(* CODESYS project CowbellCheckers_Rev8.project

Project tree, tasks and I/O mapping:
  CODESYS_SoftMotion_Win_V3 : PAC320-CXX2X-XX, Parker Hannifin, order no. PAC320-CXX2X-XX, version 3.5.9.10
    application Application
      libraries: VisuDialogs, * (System); CmpErrors, 3.3.1.40 (System); ISysTypes2, 3.5.0.0 (System); SysFile, 3.5.9.0 (System); SysTimeCore, 3.5.5.0 (System); SysTimeRtc, 3.5.5.0 (System); Util, 3.5.9.0 (System)
      task VISU_TASK (cyclic, interval 100 ms, priority 31) calls VisuElems.Visu_Prg
      task EtherCAT_Master_Sim (externalevent, external event EVENT_ECM_DC, priority 0) calls EtherCAT_Master.EtherCAT_Task [EtherCAT_Master.EtherCAT_Task], Gameplay, KingTextControl, TurnEnforcer, TestPower, MakeMove, AxisPositionFeedback, JogLogic, SetupStart, CheckForWinner, Teardown
      task FileHandler (cyclic, interval t#20ms, priority 25) calls LogData
      global variables GlobalVars
      SymbolConfiguration
      JogFunctionality/
        program JogLogic [ST]
      Visualizations/
        visualisation AreYouSure
        visualisation ErrorVis
        visualisation JogVis
        visualisation GameView
        visualisation MainView
        visualisation Congratulations
        visualisation InitScreen
        visualisation HowToPlay
        visualisation ErrorsCleared
        visualisation Checkerboard
        image pool ImagePool
        visualisation History
      axis group XYZ: TRAFO.Kin_Gantry3, axes X, Y, Z
      data type BoardSpace
      data type JumpDetail
      data type JumpProfile
      data type Piece
      global variables GVL
      GameplayFunctions/
        program boardSetup [ST]
        function assignStartingPositions [ST]
        program AxisPositionFeedback [CFC]
        function checkForJumpBlack1 [ST]
        function checkForJumpBlack2 [ST]
        function checkForJumpBlack3 [ST]
        function checkForJumpBlack4 [ST]
        function checkForJumpRed1 [ST]
        function checkForJumpRed2 [ST]
        function checkForJumpRed3 [ST]
        function checkForJumpRed4 [ST]
        function clearGlobalStack [ST]
        function clearJumpArr [ST]
        function clearPieceJumpArray [ST]
        program ClearTakenPieces [ST]
        function findPieceAtGivenLocation [ST]
        function findSelectedPiece [ST]
        program Gameplay [ST]
        program HMISequence [SFC]
        program Init [ST]
        program JumpPieces [ST]
        program KingTextControl [ST]
        program MakeJump [ST]
        program MakeMove [ST]
        function movePiece [ST]
        function block MovePieceMotion [CFC]
        function movePieceToStart [ST]
        function pieceSelect [ST]
        function placePiece [ST]
        function pop [ST]
        program ProgramFlow [SFC]
        function push [ST]
        program TestPower [CFC]
        function block timeDelay [CFC]
        program TurnEnforcer [ST]
        program UpdateValidMoveArrays [ST]
        program SetupStart [ST]
        program MoveHome [ST]
        program SetupFromStart [ST]
        program CheckForWinner [ST]
        program Teardown [ST]
        program TestMyArray [ST]
      trace Trace (task EtherCAT_Master_Sim): AxisPositionFeedback.pos.c.Z, MakeMove.moveTest.zPos
      MobileVisualizations/
        visualisation MobileVis
      data type History
      global variables PersistentVars
      function block ArrayMove [ST]
      Export/
        function GetHeaderString [ST]
        function GetLogMsgString [ST]
        function GetTimeStampString [ST]
        program LogData [ST]
        program LogWinnerNames [ST]
        program Run_FileCopy [CFC]
        function block Test_FileCopy [ST]
    SoftMotion General Axis Pool
    EtherCAT_Master : PAC320 EtherCAT Master, Parker Hannifin, order no. PAC320-XXXXX-XX, version 3.5.9.10
      PD_xxC_Standard_EtherCAT_drive_2 : PD-xxC - Standard EtherCAT drive(CoE,EoE,FoE) V2.0, Parker Hannifin, version Revision=16#00000002
          settings: DC sync0 cycletime = 4000
          unmapped channels: Controlword, Target Position, Touch Probe Function, Digital Ouputs, Statusword, Position Actual Value, Following Error Actual Value, Touch Probe Status, Touch Probe 1 Positive Edge Position Value, Digital Inputs
        Z : SM_Drive_GenericDSP402, 3S - Smart Software Solutions GmbH, order no. 0, version 4.0.0.0
            settings: wDriveID = 2; dwRatioTechUnitsDenom = 262144; iRatioTechUnitsNum = 5; fSWMaxVelocity = 100; fSWLimitPositive = 58; fSWLimitNegative = -10; bSWLimitEnable = TRUE; ScalingIncs = 262144; ScalingUnits = 5; AdrOffset_8010 = 36; BitOffset_8010 = 0; BitLength_8010 = 16; Address_8010 = '%QW18'; Type_8010 = 'UINT'; AddressPointer_8010 = ADR(%QW18); AdrOffset_8020 = 40; BitOffset_8020 = 0; BitLength_8020 = 32; Address_8020 = '%QD10'; Type_8020 = 'DINT'; AddressPointer_8020 = ADR(%QD10); AdrOffset_8030 = 4294967295; BitOffset_8030 = 0; BitLength_8030 = 0; Address_8030 = ''; Type_8030 = ''; AddressPointer_8030 = 0; AdrOffset_8040 = 4294967295; BitOffset_8040 = 0; BitLength_8040 = 0; Address_8040 = ''; Type_8040 = ''; AddressPointer_8040 = 0; AdrOffset_8050 = 4294967295; BitOffset_8050 = 0; BitLength_8050 = 0; Address_8050 = ''; Type_8050 = ''; AddressPointer_8050 = 0; AdrOffset_8060 = 44;
              BitOffset_8060 = 0; BitLength_8060 = 16; Address_8060 = '%QW22'; Type_8060 = 'UINT'; AddressPointer_8060 = ADR(%QW22); AdrOffset_8070 = 4294967295; BitOffset_8070 = 0; BitLength_8070 = 0; Address_8070 = ''; Type_8070 = ''; AddressPointer_8070 = 0; AdrOffset_8080 = 4294967295; BitOffset_8080 = 0; BitLength_8080 = 0; Address_8080 = ''; Type_8080 = ''; AddressPointer_8080 = 0; AdrOffset_8090 = 48; BitOffset_8090 = 0; BitLength_8090 = 32; Address_8090 = '%QD12'; Type_8090 = 'UDINT'; AddressPointer_8090 = ADR(%QD12); AdrOffset_8510 = 52; BitOffset_8510 = 0; BitLength_8510 = 16; Address_8510 = '%IW26'; Type_8510 = 'UINT'; AddressPointer_8510 = ADR(%IW26); AdrOffset_8520 = 56; BitOffset_8520 = 0; BitLength_8520 = 32; Address_8520 = '%ID14'; Type_8520 = 'DINT'; AddressPointer_8520 = ADR(%ID14); AdrOffset_8530 = 4294967295; BitOffset_8530 = 0; BitLength_8530 = 0; Address_8530 = ''; Type_8530 = '';
              AddressPointer_8530 = 0; AdrOffset_8540 = 4294967295; BitOffset_8540 = 0; BitLength_8540 = 0; Address_8540 = ''; Type_8540 = ''; AddressPointer_8540 = 0; AdrOffset_8550 = 4294967295; BitOffset_8550 = 0; BitLength_8550 = 0; Address_8550 = ''; Type_8550 = ''; AddressPointer_8550 = 0; AdrOffset_8560 = 72; BitOffset_8560 = 0; BitLength_8560 = 32; Address_8560 = '%ID18'; Type_8560 = 'UDINT'; AddressPointer_8560 = ADR(%ID18); AdrOffset_8570 = 64; BitOffset_8570 = 0; BitLength_8570 = 16; Address_8570 = '%IW32'; Type_8570 = 'UINT'; AddressPointer_8570 = ADR(%IW32); AdrOffset_8580 = 68; BitOffset_8580 = 0; BitLength_8580 = 32; Address_8580 = '%ID17'; Type_8580 = 'DINT'; AddressPointer_8580 = ADR(%ID17); AdrOffset_8590 = 4294967295; BitOffset_8590 = 0; BitLength_8590 = 0; Address_8590 = ''; Type_8590 = ''; AddressPointer_8590 = 0; AdrOffset_8600 = 4294967295; BitOffset_8600 = 0; BitLength_8600 = 0;
              Address_8600 = ''; Type_8600 = ''; AddressPointer_8600 = 0; AdrOffset_8600 = 4294967295; BitOffset_8600 = 0; BitLength_8600 = 0; Address_8610 = ''; Type_8610 = ''; AddressPointer_8610 = 0; AdrOffset_8620 = 60; BitOffset_8620 = 0; BitLength_8620 = 32; Address_8620 = '%ID15'; Type_8620 = 'DINT'; AddressPointer_8620 = ADR(%ID15)
      PD_xxC_Standard_EtherCAT_drive : PD-xxC - Standard EtherCAT drive(CoE,EoE,FoE) V2.0, Parker Hannifin, version Revision=16#00000002
          settings: DC sync0 cycletime = 4000
          unmapped channels: Controlword, Target Position, Touch Probe Function, Digital Ouputs, Statusword, Position Actual Value, Following Error Actual Value, Touch Probe Status, Touch Probe 1 Positive Edge Position Value, Digital Inputs
        X : SM_Drive_GenericDSP402, 3S - Smart Software Solutions GmbH, order no. 0, version 4.0.0.0
            settings: wDriveID = 3; dwRatioTechUnitsDenom = 3670016; iRatioTechUnitsNum = -125; fSWMaxVelocity = 100; fSWLimitPositive = 315; fSWLimitNegative = 0; bSWLimitEnable = TRUE; ScalingIncs = 524288; ScalingMotorTurns2 = 7; ScalingUnits = 125; InvertDirection = TRUE; AdrOffset_8010 = 4; BitOffset_8010 = 0; BitLength_8010 = 16; Address_8010 = '%QW2'; Type_8010 = 'UINT'; AddressPointer_8010 = ADR(%QW2); AdrOffset_8020 = 8; BitOffset_8020 = 0; BitLength_8020 = 32; Address_8020 = '%QD2'; Type_8020 = 'DINT'; AddressPointer_8020 = ADR(%QD2); AdrOffset_8030 = 4294967295; BitOffset_8030 = 0; BitLength_8030 = 0; Address_8030 = ''; Type_8030 = ''; AddressPointer_8030 = 0; AdrOffset_8040 = 4294967295; BitOffset_8040 = 0; BitLength_8040 = 0; Address_8040 = ''; Type_8040 = ''; AddressPointer_8040 = 0; AdrOffset_8050 = 4294967295; BitOffset_8050 = 0; BitLength_8050 = 0; Address_8050 = ''; Type_8050 = '';
              AddressPointer_8050 = 0; AdrOffset_8060 = 12; BitOffset_8060 = 0; BitLength_8060 = 16; Address_8060 = '%QW6'; Type_8060 = 'UINT'; AddressPointer_8060 = ADR(%QW6); AdrOffset_8070 = 4294967295; BitOffset_8070 = 0; BitLength_8070 = 0; Address_8070 = ''; Type_8070 = ''; AddressPointer_8070 = 0; AdrOffset_8080 = 4294967295; BitOffset_8080 = 0; BitLength_8080 = 0; Address_8080 = ''; Type_8080 = ''; AddressPointer_8080 = 0; AdrOffset_8090 = 16; BitOffset_8090 = 0; BitLength_8090 = 32; Address_8090 = '%QD4'; Type_8090 = 'UDINT'; AddressPointer_8090 = ADR(%QD4); AdrOffset_8510 = 4; BitOffset_8510 = 0; BitLength_8510 = 16; Address_8510 = '%IW2'; Type_8510 = 'UINT'; AddressPointer_8510 = ADR(%IW2); AdrOffset_8520 = 8; BitOffset_8520 = 0; BitLength_8520 = 32; Address_8520 = '%ID2'; Type_8520 = 'DINT'; AddressPointer_8520 = ADR(%ID2); AdrOffset_8530 = 4294967295; BitOffset_8530 = 0; BitLength_8530 = 0;
              Address_8530 = ''; Type_8530 = ''; AddressPointer_8530 = 0; AdrOffset_8540 = 4294967295; BitOffset_8540 = 0; BitLength_8540 = 0; Address_8540 = ''; Type_8540 = ''; AddressPointer_8540 = 0; AdrOffset_8550 = 4294967295; BitOffset_8550 = 0; BitLength_8550 = 0; Address_8550 = ''; Type_8550 = ''; AddressPointer_8550 = 0; AdrOffset_8560 = 24; BitOffset_8560 = 0; BitLength_8560 = 32; Address_8560 = '%ID6'; Type_8560 = 'UDINT'; AddressPointer_8560 = ADR(%ID6); AdrOffset_8570 = 16; BitOffset_8570 = 0; BitLength_8570 = 16; Address_8570 = '%IW8'; Type_8570 = 'UINT'; AddressPointer_8570 = ADR(%IW8); AdrOffset_8580 = 20; BitOffset_8580 = 0; BitLength_8580 = 32; Address_8580 = '%ID5'; Type_8580 = 'DINT'; AddressPointer_8580 = ADR(%ID5); AdrOffset_8590 = 4294967295; BitOffset_8590 = 0; BitLength_8590 = 0; Address_8590 = ''; Type_8590 = ''; AddressPointer_8590 = 0; AdrOffset_8600 = 4294967295;
              BitOffset_8600 = 0; BitLength_8600 = 0; Address_8600 = ''; Type_8600 = ''; AddressPointer_8600 = 0; AdrOffset_8600 = 4294967295; BitOffset_8600 = 0; BitLength_8600 = 0; Address_8610 = ''; Type_8610 = ''; AddressPointer_8610 = 0; AdrOffset_8620 = 12; BitOffset_8620 = 0; BitLength_8620 = 32; Address_8620 = '%ID3'; Type_8620 = 'DINT'; AddressPointer_8620 = ADR(%ID3)
      PD_xxC_Standard_EtherCAT_drive_1 : PD-xxC - Standard EtherCAT drive(CoE,EoE,FoE) V2.0, Parker Hannifin, version Revision=16#00000002
          settings: DC sync0 cycletime = 4000
          unmapped channels: Controlword, Target Position, Touch Probe Function, Digital Ouputs, Statusword, Position Actual Value, Following Error Actual Value, Touch Probe Status, Touch Probe 1 Positive Edge Position Value, Digital Inputs
        Y : SM_Drive_GenericDSP402, 3S - Smart Software Solutions GmbH, order no. 0, version 4.0.0.0
            settings: dwRatioTechUnitsDenom = 65536; iRatioTechUnitsNum = 3; fSWMaxVelocity = 100; fSWLimitPositive = 184; fSWLimitNegative = 0; bSWLimitEnable = TRUE; ScalingIncs = 262144; ScalingMotorTurns2 = 5; ScalingUnits = 60; AdrOffset_8010 = 20; BitOffset_8010 = 0; BitLength_8010 = 16; Address_8010 = '%QW10'; Type_8010 = 'UINT'; AddressPointer_8010 = ADR(%QW10); AdrOffset_8020 = 24; BitOffset_8020 = 0; BitLength_8020 = 32; Address_8020 = '%QD6'; Type_8020 = 'DINT'; AddressPointer_8020 = ADR(%QD6); AdrOffset_8030 = 4294967295; BitOffset_8030 = 0; BitLength_8030 = 0; Address_8030 = ''; Type_8030 = ''; AddressPointer_8030 = 0; AdrOffset_8040 = 4294967295; BitOffset_8040 = 0; BitLength_8040 = 0; Address_8040 = ''; Type_8040 = ''; AddressPointer_8040 = 0; AdrOffset_8050 = 4294967295; BitOffset_8050 = 0; BitLength_8050 = 0; Address_8050 = ''; Type_8050 = ''; AddressPointer_8050 = 0; AdrOffset_8060 = 28;
              BitOffset_8060 = 0; BitLength_8060 = 16; Address_8060 = '%QW14'; Type_8060 = 'UINT'; AddressPointer_8060 = ADR(%QW14); AdrOffset_8070 = 4294967295; BitOffset_8070 = 0; BitLength_8070 = 0; Address_8070 = ''; Type_8070 = ''; AddressPointer_8070 = 0; AdrOffset_8080 = 4294967295; BitOffset_8080 = 0; BitLength_8080 = 0; Address_8080 = ''; Type_8080 = ''; AddressPointer_8080 = 0; AdrOffset_8090 = 32; BitOffset_8090 = 0; BitLength_8090 = 32; Address_8090 = '%QD8'; Type_8090 = 'UDINT'; AddressPointer_8090 = ADR(%QD8); AdrOffset_8510 = 28; BitOffset_8510 = 0; BitLength_8510 = 16; Address_8510 = '%IW14'; Type_8510 = 'UINT'; AddressPointer_8510 = ADR(%IW14); AdrOffset_8520 = 32; BitOffset_8520 = 0; BitLength_8520 = 32; Address_8520 = '%ID8'; Type_8520 = 'DINT'; AddressPointer_8520 = ADR(%ID8); AdrOffset_8530 = 4294967295; BitOffset_8530 = 0; BitLength_8530 = 0; Address_8530 = ''; Type_8530 = '';
              AddressPointer_8530 = 0; AdrOffset_8540 = 4294967295; BitOffset_8540 = 0; BitLength_8540 = 0; Address_8540 = ''; Type_8540 = ''; AddressPointer_8540 = 0; AdrOffset_8550 = 4294967295; BitOffset_8550 = 0; BitLength_8550 = 0; Address_8550 = ''; Type_8550 = ''; AddressPointer_8550 = 0; AdrOffset_8560 = 48; BitOffset_8560 = 0; BitLength_8560 = 32; Address_8560 = '%ID12'; Type_8560 = 'UDINT'; AddressPointer_8560 = ADR(%ID12); AdrOffset_8570 = 40; BitOffset_8570 = 0; BitLength_8570 = 16; Address_8570 = '%IW20'; Type_8570 = 'UINT'; AddressPointer_8570 = ADR(%IW20); AdrOffset_8580 = 44; BitOffset_8580 = 0; BitLength_8580 = 32; Address_8580 = '%ID11'; Type_8580 = 'DINT'; AddressPointer_8580 = ADR(%ID11); AdrOffset_8590 = 4294967295; BitOffset_8590 = 0; BitLength_8590 = 0; Address_8590 = ''; Type_8590 = ''; AddressPointer_8590 = 0; AdrOffset_8600 = 4294967295; BitOffset_8600 = 0; BitLength_8600 = 0;
              Address_8600 = ''; Type_8600 = ''; AddressPointer_8600 = 0; AdrOffset_8600 = 4294967295; BitOffset_8600 = 0; BitLength_8600 = 0; Address_8610 = ''; Type_8610 = ''; AddressPointer_8610 = 0; AdrOffset_8620 = 36; BitOffset_8620 = 0; BitLength_8620 = 32; Address_8620 = '%ID9'; Type_8620 = 'DINT'; AddressPointer_8620 = ADR(%ID9)
      PAC320_BusCoupler : PAC320 BusCoupler, Parker Hannifin, version Revision=16#00000001
          settings: StationAlias = 0; DC sync0 cycletime = 4000; DC sync1 cycletime = 4000
        PACIO_DI16_DO16_1 : DI16/DO16 1ms 0.5A LS (PACIO-450-13), Parker Hannifin, version Revision=16#00000001
            settings: DC sync0 cycletime = 4000; DC sync1 cycletime = 4000
            output GripperMove : BIT  // DigitalOutput0
            unmapped channels: DigitalOutput1, DigitalOutput2, DigitalOutput3, DigitalOutput4, DigitalOutput5, DigitalOutput6, DigitalOutput7, DigitalOutput8, DigitalOutput9, DigitalOutput10, DigitalOutput11, DigitalOutput12, DigitalOutput13, DigitalOutput14, DigitalOutput15, DigitalInput0, DigitalInput1, DigitalInput2, DigitalInput3, DigitalInput4, DigitalInput5, DigitalInput6, DigitalInput7, DigitalInput8, DigitalInput9, DigitalInput10, DigitalInput11, DigitalInput12, DigitalInput13, DigitalInput14, DigitalInput15
  libraries: VisuSymbols, 3.5.8.0 (System); VisuDialogs, * (System); SM3_Basic, 4.0.0.0 (3S - Smart Software Solutions GmbH)
  text COWBELL_PROGRAMMING_STANDARD
  text list GlobalTextList
  text GameInformation
  5ce3da45-db07-42e7-a21c-a00fff4ed8f6|C:\Users\Lance\Desktop\cATCh Final Project\Project Images\LeftCheck.png
  5ce3da45-db07-42e7-a21c-a00fff4ed8f6|C:\Users\Lance\Desktop\cATCh Final Project\Project Images\LargeCheck.jpg
  5ce3da45-db07-42e7-a21c-a00fff4ed8f6|C:\Users\Lance\Desktop\cATCh Final Project\Project Images\AngleCheck.jpg
  5ce3da45-db07-42e7-a21c-a00fff4ed8f6|C:\Users\Lance\Desktop\cATCh Final Project\Project Images\AngleCheck.jpg
  5ce3da45-db07-42e7-a21c-a00fff4ed8f6|C:\Users\Lance\Desktop\cATCh Final Project\Project Images\LeftCheck.png
  5ce3da45-db07-42e7-a21c-a00fff4ed8f6|C:\Users\Lance\Desktop\cATCh Final Project\Cowbell Logo.png
  5ce3da45-db07-42e7-a21c-a00fff4ed8f6|C:\Users\Lance\Desktop\cATCh Final Project\Project Images\RedCheck.jpg
  5ce3da45-db07-42e7-a21c-a00fff4ed8f6|C:\Users\Lance\Desktop\cATCh Final Project\Project Images\MedCheck_edited.jpg
  5ce3da45-db07-42e7-a21c-a00fff4ed8f6|C:\Users\Lance\Desktop\cATCh Final Project\Project Images\MedCheck.jpg
  5ce3da45-db07-42e7-a21c-a00fff4ed8f6|C:\Users\Lance\Desktop\cATCh Final Project\Project Images\RedCheck.jpg
  5ce3da45-db07-42e7-a21c-a00fff4ed8f6|C:\Users\Lance\Desktop\cATCh Final Project\Project Images\RightCheck.jpg
  5ce3da45-db07-42e7-a21c-a00fff4ed8f6|C:\Users\Lance\Desktop\cATCh Final Project\Project Images\MedCheck_edited.jpg
  5ce3da45-db07-42e7-a21c-a00fff4ed8f6|C:\Users\Lance\Desktop\AreYouSurePic.png
*)

// CODESYS_SoftMotion_Win_V3/Application/BoardSpace
TYPE BoardSpace :
STRUCT
	isBlack : BOOL := FALSE;
	isRed : BOOL := FALSE;
	isEmpty : BOOL := TRUE;
	chosenForMove : BOOL := FALSE;
	
	xLoc : INT;
END_STRUCT
END_TYPE

// CODESYS_SoftMotion_Win_V3/Application/JumpDetail
TYPE JumpDetail :
STRUCT
	
	xMoveLocation : INT := -1;
	yMoveLocation : INT := -1;
	jumpedColor : INT := -1;
	jumpedIndex : INT := -1;
	
	
END_STRUCT
END_TYPE

// CODESYS_SoftMotion_Win_V3/Application/JumpProfile
TYPE JumpProfile :
STRUCT
	jumpRef : INT;
	lastJumpRef : INT := -1;
	xMoveLocation : INT;
	yMoveLocation : INT;
	xJumpedLocation : INT;
	yJumpedLocation : INT;
	numPiecesToJump : INT;
	jumpedPieceColor : INT;
	jumpedPieceIndex : INT;
	jumpingPieceX : INT;
	jumpingPieceY : INT;
END_STRUCT
END_TYPE

// CODESYS_SoftMotion_Win_V3/Application/Piece
TYPE Piece :
STRUCT
	isBlack : BOOL := FALSE; // False indicates that a piece is red; true indicates black
	isTaken : BOOL := FALSE; // False indicates that a piece is still in play
	isKing : BOOL := FALSE; // True indicates that a piece is a king
	isSelected : BOOL := FALSE;
	oldLocation : ARRAY [0..1] OF INT := [0,0];
	currentLocation : ARRAY [0..1] OF INT := [0,0]; // -1, -1 indicated that the piece has been taken
	translatedLocation : ARRAY [0..1] OF INT; // translated movement in terms of HMI coordinates
	startingLocation : ARRAY [0..1] OF INT;
	validMoveArr : ARRAY [0..7,0..7] OF BOOL; // 2D array represents the board, true indicates that a piece can move to that space 
	
	jumpArr : ARRAY [0..20,0..3] OF JumpDetail;
	
	startStack : INT;
	jumpedPieceIndex : INT;
	kingText : WSTRING := "";
END_STRUCT
END_TYPE

// CODESYS_SoftMotion_Win_V3/Application/History
TYPE History :
STRUCT
	
	Names: STRING;
	Moves: INT;
	
END_STRUCT
END_TYPE

// CODESYS_SoftMotion_Win_V3/Application/GlobalVars
{attribute 'qualified_only'}
(* COWBELL GLOBAL VARIABLES *)
VAR_GLOBAL
	systemEnable : BOOL;
	
	p1CheckerColor: DWORD := 16#FF000000; // 16# - interpret as hexidecimal, FF - transparency (Fully Opaque, 00 fully transparent), FF - Red, FF - Green, FF - Blue
	p2CheckerColor: DWORD := 16#FFFF0000;
	
	p1DefaultName: STRING := 'Player_1';
	p2DefaultName: STRING := 'Player_2';
	p1Name: STRING;
	p2Name: STRING;
	winnerName: STRING;
	winnerMoves : INT;
	
	funnyText: STRING := 'Dont poke me';
	funnyCounter: INT := 0;
	
	
(***** X AXIS PARAMETERS *****)
		
	xVel: INT := 10;
	xAcc: INT := 100;
	xDec: INT := 100;
	xJerk: INT := 100;
	
	xJogFwd: BOOL;
	xJogRev: BOOL;
	
(***** Y AXIS PARAMETERS *****)
	
	yVel: INT := 10;
	yAcc: INT := 100;
	yDec: INT := 100;
	yJerk: INT := 100;
	
	yJogFwd: BOOL;
	yJogRev: BOOL;
	
(***** Z AXIS PARAMETERS *****)
	
	zVel: INT := 10;
	zAcc: INT := 100;
	zDec: INT := 100;
	zJerk: INT := 100;
	
	zJogFwd: BOOL;
	zJogRev: BOOL;
	
END_VAR

// CODESYS_SoftMotion_Win_V3/Application/GVL
{attribute 'qualified_only'}
VAR_GLOBAL
	selectedPieceValidMoveArr : ARRAY [0..7,0..7] OF BOOL;
	noValidMoveArr : ARRAY [0..7,0..7] OF BOOL;
	selectedPieceValidJumpArr : ARRAY [0..7,0..7] OF BOOL;
	board : ARRAY [0..7,0..7] OF BoardSpace; // represents every space on the board
	pieces : ARRAY [0..1,0..11] OF Piece; // 1,x is any black piece, 0,x is any red piece
	redsTurn : BOOL := TRUE;
	
	homeAxes : BOOL;
	
	mechanicalSetup : BOOL;
	
	redWins : BOOL;
	blackWins : BOOL;
	
	teardown : BOOL;
	
	export : BOOL;
	
	currentRedStack : INT := 2;
	currentRedStackPos : INT := 4;
	
	currentBlackStack : INT := 2;
	currentBlackStackPos : INT := 4;
	
	jumpMoveArr : ARRAY[0..100] OF JumpProfile;
	currentJumpRef : INT := 0;
	
	xMoveSpace : INT := -1;
	yMoveSpace : INT := -1;
	
	boardIsSetup : BOOL;
	
	takenList : ARRAY [0..20,0..1] OF INT := [-1, -1,-1,-1,-1,-1,-1,-1,-1,-1,-1,-1,-1,-1,-1,-1,-1,-1,-1,-1,-1,-1,-1,-1,-1,-1,-1,-1,-1,-1,-1,-1,-1,-1,-1,-1,-1,-1,-1];
	takenListLength : INT;
	emptyTakenList : ARRAY [0..20,0..1] OF INT := [-1, -1,-1,-1,-1,-1,-1,-1,-1,-1,-1,-1,-1,-1,-1,-1,-1,-1,-1,-1,-1,-1,-1,-1,-1,-1,-1,-1,-1,-1,-1,-1,-1,-1,-1,-1,-1,-1,-1];
	
	jumpStack : ARRAY[0..3] OF JumpDetail;
	currentStackIndex : INT;
	currentJumpProfileNum : INT;
	
	emptyJumpArr : ARRAY [0..20,0..3] OF JumpDetail;
	
	redStack0Offset : ARRAY [0..1] OF INT := [0,128]; // coordinate offset of red stacks in HMI (at beginning of game)
	redStack1Offset : ARRAY [0..1] OF INT := [128,128]; // coordinate offset of red stacks in HMI (at beginning of game)
	redStack2Offset : ARRAY [0..1] OF INT := [256, 128]; // coordinate offset of red stacks in HMI (at beginning of game)
	
	blackStack0Offset : ARRAY [0..1] OF INT := [448,-576];
	blackStack1Offset : ARRAY [0..1] OF INT := [320,-576];
	blackStack2Offset : ARRAY [0..1] OF INT := [192,-576];
	
	redPiecesTaken : INT := 0;
	blackPiecesTaken : INT := 0;
	
	test : BOOL := FALSE;
	
	gameReset : BOOL := FALSE;
	
END_VAR

// CODESYS_SoftMotion_Win_V3/Application/PersistentVars
{attribute 'qualified_only'}
VAR_GLOBAL PERSISTENT RETAIN
	MyArray : ARRAY [1..20] OF History;
END_VAR

// CODESYS_SoftMotion_Win_V3/Application/GameplayFunctions/Gameplay
PROGRAM Gameplay
VAR
	//selectedPieceValidMoveArr : ARRAY [0..7,0..7] OF BOOL;
	//noValidMoveArr : ARRAY [0..7,0..7] OF BOOL;
	//board : ARRAY [0..7,0..7] OF BoardSpace; // represents every space on the board
	//pieces : ARRAY [0..1,0..11] OF Piece; // 0,x is any black piece, 1,x is any red piece
	startingPositionsRed : ARRAY [0..1,0..11] OF INT;
	startingPositionsBlack : ARRAY [0..1,0..11] OF INT;
	redIsAssigned : BOOL := FALSE;
	blackIsAssigned : BOOL := FALSE;
	
	// ****************VARIABLES FOR BOARD SETUP*******************
	numStacks : INT := 3;
	numPiecesInStack : INT := 5;
	numPieces : INT := 12;
	currentStack : INT := 0; // stack that gripper is currently drawing from
	currentPiece : INT := 0; // piece number that gripper has set up
	currentStackPos : INT := 0;	// stack position flows 0-4 from top to bottom
	currentSpace : ARRAY [0..1] OF INT;
	piecePosition : ARRAY[0..1] OF INT;
	
	done : BOOL;
	i : INT := 0;
	j : INT := 0;
	boardCleared : BOOL := FALSE;
	y: INT;
	pieceNum: INT;
	x: INT;
	temp : INT;
	commenceSetup : BOOL := FALSE; // Variable toggled by pushing the set up board button
	xPos: INT;
	yPos: INT;
	found : BOOL := FALSE;
END_VAR

IF(commenceSetup) THEN
	IF(NOT GVL.boardIsSetup) THEN
	

		// Assigns starting positions for red and black GVL.pieces
	IF(NOT redIsAssigned) THEN
		startingPositionsRed := assignStartingPositions(startingPositionsRed, TRUE);
		redIsAssigned := TRUE;
	END_IF
	IF(NOT blackIsAssigned) THEN
		startingPositionsBlack := assignStartingPositions(startingPositionsBlack, FALSE);
		blackIsAssigned := TRUE;
	END_IF


	// initializes values for red GVL.pieces
	FOR i := 0 TO (numPieces - 1) DO
		GVL.pieces[0,i].isBlack := FALSE;
		GVL.pieces[0,i].isKing := FALSE;
		GVL.pieces[0,i].isTaken := FALSE;
		GVL.pieces[0,i].currentLocation[0] := startingPositionsRed[0,i]; 
		GVL.pieces[0,i].currentLocation[1] := startingPositionsRed[1,i];
		GVL.pieces[0,i].jumpedPieceIndex := i;
		IF(i < numPiecesInStack) THEN
			GVL.pieces[0,i].startStack := 0;
		ELSIF(i < (numPiecesInStack * 2) AND i >= numPiecesInStack) THEN
			GVL.pieces[0,i].startStack := 1;
		ELSE
			GVL.pieces[0,i].startStack := 2;
		END_IF
		GVL.pieces[0,i] := movePieceToStart(GVL.pieces[0,i]);
		GVL.board[GVL.pieces[0,i].currentLocation[0], GVL.pieces[0,i].currentLocation[1]].isRed := TRUE;
		GVL.board[GVL.pieces[0,i].currentLocation[0], GVL.pieces[0,i].currentLocation[1]].isBlack := FALSE;
		GVL.board[GVL.pieces[0,i].currentLocation[0], GVL.pieces[0,i].currentLocation[1]].isEmpty := FALSE;
	END_FOR


	// initializes values for black GVL.pieces
	FOR i := 0 TO (numPieces - 1) DO
		GVL.pieces[1,i].isBlack := TRUE;
		GVL.pieces[1,i].isKing := FALSE;
		GVL.pieces[1,i].isTaken := FALSE;
		GVL.pieces[1,i].currentLocation[0] := startingPositionsBlack[0,i];
		GVL.pieces[1,i].currentLocation[1] := startingPositionsBlack[1,i];
		IF(i < numPiecesInStack) THEN
			GVL.pieces[1,i].startStack := 0;
		ELSIF(i < (numPiecesInStack * 2) AND i >= numPiecesInStack) THEN
			GVL.pieces[1,i].startStack := 1;
		ELSE
			GVL.pieces[1,i].startStack := 2;
		END_IF
		GVL.pieces[1,i] := movePieceToStart(GVL.pieces[1,i]);
		GVL.board[GVL.pieces[1,i].currentLocation[0], GVL.pieces[1,i].currentLocation[1]].isRed := FALSE;
		GVL.board[GVL.pieces[1,i].currentLocation[0], GVL.pieces[1,i].currentLocation[1]].isBlack := TRUE;
		GVL.board[GVL.pieces[1,i].currentLocation[0], GVL.pieces[1,i].currentLocation[1]].isEmpty := FALSE;
	END_FOR

	GVL.boardIsSetup := TRUE;
END_IF

// Setup valid moves for red
FOR i:= 0 TO numPieces - 1 DO
	x:= GVL.pieces[0,i].currentLocation[0];
	y := GVL.pieces[0,i].currentLocation[1];
	
	// Checks for move up and right
	IF(x+1 < 8 AND y+1 < 8 AND GVL.board[x+1,y+1].isEmpty) THEN
		GVL.pieces[0,i].validMoveArr[x+1,y+1] := TRUE;
	END_IF

	// Checks for move up and left
	IF(x-1 >= 0 AND y+1 < 8 AND GVL.board[x-1,y+1].isEmpty) THEN
		GVL.pieces[0,i].validMoveArr[x-1,y+1] := TRUE;
	END_IF
	
	IF(x+1 < 8 AND y+1 < 8 AND NOT GVL.board[x+1,y+1].isEmpty AND GVL.board[x+1,y+1].isBlack) THEN
		
		//possible jump
	END_IF
	
END_FOR

// Setup valid moves for black
FOR i:= 0 TO numPieces - 1 DO
	x:= GVL.pieces[1,i].currentLocation[0];
	y := GVL.pieces[1,i].currentLocation[1];
	
	// Checks for move up and right
	IF(x+1 < 8 AND y+1 < 8 AND GVL.board[x+1,y-1].isEmpty) THEN
		GVL.pieces[1,i].validMoveArr[x+1,y-1] := TRUE;
	END_IF

	// Checks for move up and left
	IF(x-1 >= 0 AND y+1 < 8 AND GVL.board[x-1,y-1].isEmpty) THEN
		GVL.pieces[1,i].validMoveArr[x-1,y-1] := TRUE;
	END_IF
	
	(*
	IF(x+1 < 8 AND y+1 < 8 AND NOT GVL.board[x+1,y+1].isEmpty AND GVL.board[x+1,y+1].isBlack) THEN
		
		//possible jump
	END_IF
	*)
	
END_FOR

GVL.mechanicalSetup := TRUE;


END_IF

END_PROGRAM

// CODESYS_SoftMotion_Win_V3/Application/GameplayFunctions/assignStartingPositions
FUNCTION assignStartingPositions : ARRAY [0..1,0..11] OF INT;
VAR_INPUT
	startingPos : ARRAY [0..1,0..11] OF INT;
	isRed : BOOL;
END_VAR
VAR
	numPieces : INT := 12;
	
	i: INT;
	y: INT;
	x: INT;
	temp: INT;
END_VAR

IF(isRed) THEN
	FOR i := 0 TO (numPieces - 1) DO 	
		y := i / 4;
		x := ((2 * i) MOD 8) + (y MOD 2);
		startingPos[0,i] := x;
		startingPos[1,i] := y;
	END_FOR
ELSE
	FOR i := 0 TO (numPieces - 1) DO 
		temp := i / 4;
		x := ((2 * i) MOD 8) + (temp MOD 2);
		y := temp + 5;
		x := x + 1;
		IF(x >= 8) THEN
			x := x MOD 8;
		END_IF
		startingPos[0,i] := x;
		startingPos[1,i] := y;	
	END_FOR
END_IF

assignStartingPositions := startingPos;
RETURN;

END_FUNCTION

// CODESYS_SoftMotion_Win_V3/Application/GameplayFunctions/movePieceToStart
FUNCTION movePieceToStart : Piece
VAR_INPUT
	currentPiece : Piece;
END_VAR
VAR
	
	spaceTranslation : ARRAY [0..1] OF INT; // small numbers (0-7) that indicate how many spaces a piece needs to be moved
	sizeOfMoveX : INT := 64;
	sizeOfMoveY : INT := -64;
END_VAR

movePieceToStart := currentPiece;
IF(NOT movePieceToStart.isBlack) THEN
	// Moves pieces from their stack to the origin (board sqaure 0,0 or bottom left corner)
	IF(currentPiece.startStack = 0) THEN
		movePieceToStart.translatedLocation[0] := currentPiece.translatedLocation[0] - GVL.redStack0Offset[0];
		movePieceToStart.translatedLocation[1] := currentPiece.translatedLocation[1] - GVL.redStack0Offset[1];
		
	ELSIF(currentPiece.startStack = 1) THEN
		movePieceToStart.translatedLocation[0] := currentPiece.translatedLocation[0] - GVL.redStack1Offset[0];
		movePieceToStart.translatedLocation[1] := currentPiece.translatedLocation[1] - GVL.redStack1Offset[1];
	ELSE
		movePieceToStart.translatedLocation[0] := currentPiece.translatedLocation[0] - GVL.redStack2Offset[0];
		movePieceToStart.translatedLocation[1] := currentPiece.translatedLocation[1] - GVL.redStack2Offset[1];
	END_IF
ELSE
	IF(currentPiece.startStack = 0) THEN
		movePieceToStart.translatedLocation[0] := currentPiece.translatedLocation[0] - GVL.blackStack0Offset[0];
		movePieceToStart.translatedLocation[1] := currentPiece.translatedLocation[1] - GVL.blackStack0Offset[1];
	ELSIF(currentPiece.startStack = 1) THEN
		movePieceToStart.translatedLocation[0] := currentPiece.translatedLocation[0] - GVL.blackStack1Offset[0];
		movePieceToStart.translatedLocation[1] := currentPiece.translatedLocation[1] - GVL.blackStack1Offset[1];
	ELSE
		movePieceToStart.translatedLocation[0] := currentPiece.translatedLocation[0] - GVL.blackStack2Offset[0];
		movePieceToStart.translatedLocation[1] := currentPiece.translatedLocation[1] - GVL.blackStack2Offset[1];
	END_IF			

END_IF

movePieceToStart.startingLocation := movePieceToStart.translatedLocation;

spaceTranslation[0] := movePieceToStart.currentLocation[0] - movePieceToStart.oldLocation[0];
spaceTranslation[1] := movePieceToStart.currentLocation[1] - movePieceToStart.oldLocation[1];

movePieceToStart.translatedLocation[0] := movePieceToStart.translatedLocation[0] + (spaceTranslation[0] * sizeOfMoveX);
movePieceToStart.translatedLocation[1] := movePieceToStart.translatedLocation[1] + (spaceTranslation[1] * sizeOfMoveY);

// set oldLocation to currentLocation
movePieceToStart.oldLocation[0] := movePieceToStart.currentLocation[0];
movePieceToStart.oldLocation[1] := movePieceToStart.currentLocation[1];


RETURN;

END_FUNCTION

// CODESYS_SoftMotion_Win_V3/Application/GameplayFunctions/KingTextControl
PROGRAM KingTextControl
VAR
	i : INT;
END_VAR

FOR i := 0 TO 11 DO
	IF(GVL.pieces[0,i].isKing) THEN
		GVL.pieces[0,i].kingText := "K";
	END_IF
	IF(GVL.pieces[1,i].isKing) THEN
		GVL.pieces[1,i].kingText := "K";
	END_IF
END_FOR

END_PROGRAM

// CODESYS_SoftMotion_Win_V3/Application/GameplayFunctions/TurnEnforcer
PROGRAM TurnEnforcer
VAR
	i : INT;
	wrongColorSelected : BOOL;
END_VAR

// Stops user from selecting a piece that is taken
FOR i := 0 TO 11 DO
	IF(GVL.pieces[1,i].isTaken)THEN 
		GVL.pieces[1,i].isSelected := FALSE;
	ELSIF(GVL.pieces[0,i].isTaken) THEN
		GVL.pieces[0,i].isSelected := FALSE;
	END_IF
END_FOR

// Stops user from picking the wrong color
wrongColorSelected := FALSE;

IF(GVL.redsTurn) THEN
	FOR i := 0 TO 11 DO
		IF(GVL.pieces[1,i].isSelected)THEN 
			 GVL.pieces[1,i].isSelected := FALSE;
			 wrongColorSelected := TRUE;
		END_IF
	END_FOR
ELSE
	FOR i := 0 TO 11 DO
		IF(GVL.pieces[0,i].isSelected)THEN 
			 GVL.pieces[0,i].isSelected := FALSE;
			 wrongColorSelected := TRUE;
		END_IF				
	END_FOR
END_IF

IF(wrongColorSelected) THEN
	GVL.selectedPieceValidMoveArr := GVL.noValidMoveArr;
END_IF

END_PROGRAM

// CODESYS_SoftMotion_Win_V3/Application/GameplayFunctions/TestPower
PROGRAM TestPower

VAR_INPUT
	systemReset: BOOL;
END_VAR

VAR
	xReset: MC_Reset;
	xJogMove: MC_Jog;
	
	yReset: MC_Reset;
	yJogMove: MC_Jog;
	
	zJogMove: MC_Jog;
	zReset: MC_Reset;
	
	xPower: MC_Power;
	yPower: MC_Power;
	zPower: MC_Power;
	
	EnableAxes: MC_GroupEnable;
	Enable: BOOL;
	GroupEnable: BOOL;
END_VAR

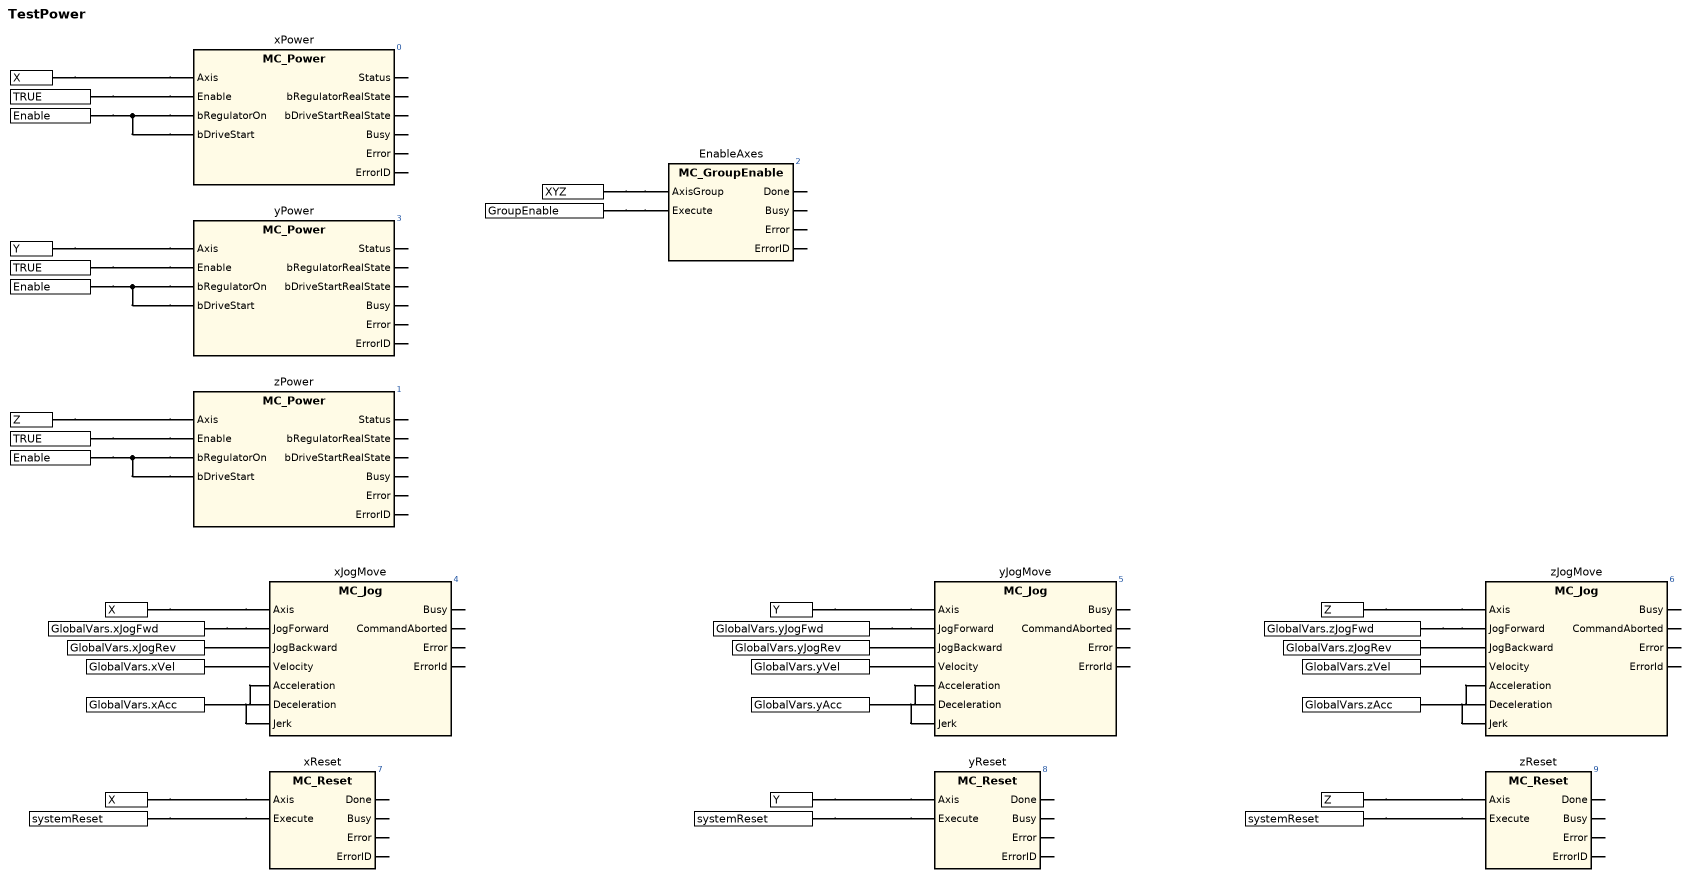
xPower(Axis := X, Enable := TRUE, bRegulatorOn := Enable, bDriveStart := Enable); // MC_Power
zPower(Axis := Z, Enable := TRUE, bRegulatorOn := Enable, bDriveStart := Enable); // MC_Power
EnableAxes(AxisGroup := XYZ, Execute := GroupEnable); // MC_GroupEnable
yPower(Axis := Y, Enable := TRUE, bRegulatorOn := Enable, bDriveStart := Enable); // MC_Power
xJogMove(
    Axis := X,
    JogForward := GlobalVars.xJogFwd,
    JogBackward := GlobalVars.xJogRev,
    Velocity := GlobalVars.xVel,
    Acceleration := GlobalVars.xAcc,
    Deceleration := GlobalVars.xAcc,
    Jerk := GlobalVars.xAcc); // MC_Jog
yJogMove(
    Axis := Y,
    JogForward := GlobalVars.yJogFwd,
    JogBackward := GlobalVars.yJogRev,
    Velocity := GlobalVars.yVel,
    Acceleration := GlobalVars.yAcc,
    Deceleration := GlobalVars.yAcc,
    Jerk := GlobalVars.yAcc); // MC_Jog
zJogMove(
    Axis := Z,
    JogForward := GlobalVars.zJogFwd,
    JogBackward := GlobalVars.zJogRev,
    Velocity := GlobalVars.zVel,
    Acceleration := GlobalVars.zAcc,
    Deceleration := GlobalVars.zAcc,
    Jerk := GlobalVars.zAcc); // MC_Jog
xReset(Axis := X, Execute := systemReset); // MC_Reset
yReset(Axis := Y, Execute := systemReset); // MC_Reset
zReset(Axis := Z, Execute := systemReset); // MC_Reset

END_PROGRAM

// CODESYS_SoftMotion_Win_V3/Application/GameplayFunctions/MakeMove
PROGRAM MakeMove
// AUTHOR: Ahren Young
// This code will run continuously throughout the life of the program. The purpose of this code
// is to handle moving, jumping and taking of pieces. All actions associated with these actions
// will be handled in this code.
// Transition from cases flows top to bottom, and is done so that the movement code at the end
// of the case statement will always run in order to ensure complete motion.
// 
// moveSpace variables are only changed when a square is pushed in the HMI
// A move will only be excuted when the a square is pushed that is a valid move
// for the piece that is selected by the current user (i.e. the piece is highlighted
// in the HMI
VAR
	i : INT;
	counter : INT;
	xCurrentSpace : INT;
	yCurrentSpace : INT;
	currentPiece : Piece;
	selected : BOOL;
	redOrBlack : INT;
	jumpedPieceIndex : INT;
	
	spaceTranslation : ARRAY [0..1] OF INT; // small numbers (0-7) that indicate how many spaces a piece needs to be moved
	sizeOfMoveX : INT := 64; // Space on the HMI that a piece must be translated
	sizeOfMoveY : INT := -64; // Space on the HMI that a piece must be translated
	
	caseState : INT := 000;
	moveTest : MovePieceMotion;
	
	spaceOffset : LREAL := 20;
	xOffset : LREAL := 79.9;
	yOffset : LREAL := 18.3;
	zUp : LREAL := 0;
	zDown: LREAL := 55;
	
	blackStackXOffset : LREAL := 260.2;
	blackStackYOffset : LREAL := 159.8;
	
	redStackXOffset : LREAL := 32.1;
	redStackYOffset : LREAL := 159.8;
	
	stackXDistApart : LREAL := 0;
	stackYDistApart : LREAL := -70;
	
	
	pieceOffset : LREAL := 6.2;
	(*
	currentRedStack : INT := 2;
	currentRedStackPos : INT := 4;
	
	currentBlackStack : INT := 2;
	currentBlackStackPos : INT := 4;
	*)
	selectedPiece : ARRAY [0..1] OF INT;
	
	xPiece: INT;
	yPiece: INT;
	
	wait : timeDelay;
	
	jumpCounter : INT; // counts how many jumps have been made and is compared to the number of jumps expected
	
	kingCurrentPiece : BOOL;
END_VAR

CASE caseState OF

// Will run in this case as long as a move space isn't selected
000:
	IF(GVL.xMoveSpace <> -1 AND GVL.yMoveSpace <> -1) THEN
		caseState := 001;
	END_IF
	
// If the move is valid, execution of the move begins by positioning
// the gripper over the piece that is to be moved
// If the move is invalid, case statement jumps back to case 000
001: 
	selectedPiece := findSelectedPiece();
	IF(GVL.selectedPieceValidMoveArr[GVL.xMoveSpace, GVL.yMoveSpace]) THEN
		xPiece := GVL.pieces[selectedPiece[0],selectedPiece[1]].currentLocation[0];
		yPiece := GVL.pieces[selectedPiece[0],selectedPiece[1]].currentLocation[1];
	
		moveTest.xPos := xOffset + (xPiece * spaceOffset);
		moveTest.yPos := yOffset + (yPiece * spaceOffset);
		moveTest.zPos := zUp;
	
		caseState := 002;
	ELSE
		// Deselects all pieces
		FOR i:=0 TO 11 DO
			GVL.pieces[0,i].isSelected := FALSE;
			GVL.pieces[1,i].isSelected := FALSE;			
		END_FOR
		GVL.xMoveSpace := -1;
		GVL.yMoveSpace := -1;
		
		caseState := 000;
	END_IF

// Move is executed	
002:
	moveTest.ExecuteMove := TRUE;
	caseState := 003;

// Once the gripper is in position above the piece to be moved
// execute move is set to false
003:
	IF(moveTest.MoveDone) THEN
		caseState := 004;
		moveTest.ExecuteMove := FALSE;
	END_IF

// Sets gripper to down position over the current piece
004:
	moveTest.zPos := zDown;
	caseState := 005;

// Move is executed
005:
	moveTest.ExecuteMove := TRUE;
	caseState := 006;

// Piece is picked up and the wait is implemented so that
// the gripper is fully closed before it begins to lift up	
006:
	IF(moveTest.MoveDone)THEN
		caseState := 007;
		moveTest.ExecuteMove := FALSE;
		GripperMove := TRUE;
		wait.startTimer := TRUE;
	END_IF

// Piece has been grabbed and the gripper moves straight up
007:
	IF(wait.done) THEN
		wait.startTimer := FALSE;
		moveTest.zPos := zUp;
		caseState := 008;
	END_IF
	
// Move is executed
008: 
	moveTest.ExecuteMove := TRUE;
	caseState := 009;

// Move is completed
009:
	IF(moveTest.MoveDone)THEN
		caseState := 010;
		moveTest.ExecuteMove := FALSE;
	END_IF
	
// All actions associated with a valid move are calculated (i.e. where to move, what to jump, etc.)
// Position is set to above the space to be moved to and the piece is still in the gripper
010:
	IF(GVL.xMoveSpace >= 0 AND GVL.yMoveSpace >= 0) THEN
		selected := FALSE;
		i := 0;
		// Figure out which piece is selected
		WHILE(i < 12 AND NOT selected) DO
		
			IF(GVL.pieces[0,i].isSelected) THEN
				xCurrentSpace := GVL.pieces[0,i].currentLocation[0];
				yCurrentSpace := GVL.pieces[0,i].currentLocation[1];
				currentPiece := GVL.pieces[0,i];
				redOrBlack := 0;
				jumpedPieceIndex := i;
				selected := TRUE;
			END_IF
			IF(GVL.pieces[1,i].isSelected) THEN
				xCurrentSpace := GVL.pieces[1,i].currentLocation[0];
				yCurrentSpace := GVL.pieces[1,i].currentLocation[1];
				currentPiece := GVL.pieces[1,i];
				redOrBlack := 1;
				jumpedPieceIndex := i;
				selected := TRUE;
			END_IF
			i := i + 1;
	
		END_WHILE
	
		// Determine if the move is legal
		IF(GVL.selectedPieceValidMoveArr[GVL.xMoveSpace, GVL.yMoveSpace])THEN 
			// Perform the move
			currentPiece.translatedLocation[0] := currentPiece.startingLocation[0] + (GVL.xMoveSpace * sizeOfMoveX);
			currentPiece.translatedLocation[1] := currentPiece.startingLocation[1] + (GVL.yMoveSpace * sizeOfMoveY);;
		
		
			moveTest.xPos := xOffset + (GVL.xMoveSpace * 20);
			moveTest.yPos := yOffset + (GVL.yMoveSpace * 20);
			moveTest.zPos := zUp;

			caseState := 020;
		
		
			// sets pieces current location as the old location, as it is about to move
			currentPiece.oldLocation[0] := currentPiece.currentLocation[0];
			currentPiece.oldLocation[1] := currentPiece.currentLocation[1];
	
			// updates the current location after the move has been completed
			currentPiece.currentLocation[0] := GVL.xMoveSpace;
			currentPiece.currentLocation[1] := GVL.yMoveSpace;
		
			// Piece is red and has achieved king status
			IF(currentPiece.currentLocation[1] = 7 AND NOT currentPiece.isBlack) THEN
				currentPiece.isKing := TRUE;
				kingCurrentPiece := TRUE;
			// Piece is black and has achieved king status
			ELSIF(currentPiece.currentLocation[1] = 0 AND currentPiece.isBlack) THEN
				currentPiece.isKing := TRUE;
				kingCurrentPiece := TRUE;
			END_IF
			
		
			// updates board space player just moved from
			GVL.board[currentPiece.oldLocation[0], currentPiece.oldLocation[1]].isEmpty := TRUE;
			GVL.board[currentPiece.oldLocation[0], currentPiece.oldLocation[1]].isBlack := FALSE;
			GVL.board[currentPiece.oldLocation[0], currentPiece.oldLocation[1]].isRed := FALSE;
		
			// updates board space that the player just moved to
			GVL.board[currentPiece.currentLocation[0], currentPiece.currentLocation[1]].isEmpty := FALSE;
			IF(currentPiece.isBlack)THEN
				GVL.board[currentPiece.currentLocation[0], currentPiece.currentLocation[1]].isBlack := TRUE;
				GVL.board[currentPiece.currentLocation[0], currentPiece.currentLocation[1]].isRed := FALSE;
			ELSE
				GVL.board[currentPiece.currentLocation[0], currentPiece.currentLocation[1]].isBlack := FALSE;
				GVL.board[currentPiece.currentLocation[0], currentPiece.currentLocation[1]].isRed := TRUE;
			END_IF
		
			GVL.pieces[redOrBlack, jumpedPieceIndex] := currentPiece;
		
		
		
			// Make it the other persons turn
			IF(GVL.redsTurn) THEN
				GVL.redsTurn := FALSE;
				GlobalVars.winnerMoves := GlobalVars.winnerMoves + 1;
			ELSE
				GVL.redsTurn := TRUE;	
			END_IF
		
		
			MakeJump();
			UpdateValidMoveArrays();
		
			// Deselects all pieces
			GVL.selectedPieceValidMoveArr := GVL.noValidMoveArr;
			FOR i:=0 TO 11 DO
				GVL.pieces[0,i].isSelected := FALSE;
				GVL.pieces[1,i].isSelected := FALSE;			
			END_FOR
		
			IF(currentPiece.oldLocation[0] + 1 = currentPiece.currentLocation[0] OR
				currentPiece.oldLocation[1] + 1 = currentPiece.currentLocation[1] OR
				currentPiece.oldLocation[0] - 1 = currentPiece.currentLocation[0] OR
				currentPiece.oldLocation[1] - 1 = currentPiece.currentLocation[1]) THEN
				// DO NOTHING
			ELSE
				ClearTakenPieces();
			END_IF
		
		
		ELSE
			// Deselects all pieces
			GVL.selectedPieceValidMoveArr := GVL.noValidMoveArr;
			FOR i:=0 TO 11 DO
				GVL.pieces[0,i].isSelected := FALSE;
				GVL.pieces[1,i].isSelected := FALSE;			
			END_FOR
			
			GVL.xMoveSpace := -1;
			GVL.yMoveSpace := -1;
		
			caseState := 000;
			
		END_IF
		clearJumpArr();
		
		GVL.xMoveSpace := -1;
		GVL.yMoveSpace := -1;

		GVL.currentJumpRef := 0;

		//counter := counter + 1;
		

		

			
	END_IF
	
// Move is executed
020:
	moveTest.ExecuteMove := TRUE;
	caseState := 030;
	
// Move is completed
030:
	IF(moveTest.MoveDone) THEN
		caseState := 031;
		moveTest.ExecuteMove := FALSE;
		UpdateValidMoveArrays();
	END_IF
	

// Sets gripper to down position over the space where the piece is to be moved
031:
	moveTest.zPos := zDown;
	caseState := 032;
	
// Move is executed
032:
	moveTest.ExecuteMove := TRUE;
	caseState := 033;

// Move execution is completed
// Gripper is opened and the piece is dropped off at its location
// A wait is implemented to ensure accuracy
033:	
	IF(moveTest.MoveDone)THEN
		caseState := 034;
		moveTest.ExecuteMove := FALSE;
		GripperMove := FALSE;
		wait.startTimer := TRUE;
	END_IF
	
// Sets gripper to up position over the current piece
034:
	IF(wait.done)THEN
		wait.startTimer := FALSE;
		moveTest.zPos := zUp;
		caseState := 035;
	END_IF
	
// Move is executed
035:
	moveTest.ExecuteMove := TRUE;
	caseState := 036;

// Moving the current piece has been completed
// next any pieces that are set to be taken based on being jumped will be taken
// jumpCounter is set to 0 as that is the number of jumps that have been performed
// it is already known how many jumps are expected to be performed
036:	
	IF(moveTest.MoveDone)THEN
		caseState := 040;
		moveTest.ExecuteMove := FALSE;
		jumpCounter := 0;	
	END_IF
	
	
// Moves over the top of the piece to be jumped
// If no pieces are set to be jumped, jump to case 070, where kinging is performed
040:
	IF(jumpCounter < GVL.takenListLength) THEN
		xPiece := GVL.takenList[jumpCounter,0];
		yPiece := GVL.takenList[jumpCounter,1];
		IF(xPiece >= 0)THEN
			moveTest.xPos := xOffset + (xPiece * spaceOffset);
			moveTest.yPos := yOffset + (yPiece * spaceOffset);
			moveTest.zPos := zUp;
			caseState := 041;
		ELSE
			caseState := 070;
		END_IF
	ELSE
		caseState := 070;	
	END_IF
	
// Move is executed
041:
	moveTest.ExecuteMove := TRUE;
	caseState := 042;
	
// Move is completed
042:
	IF(moveTest.MoveDone) THEN
		caseState := 043;
		moveTest.ExecuteMove := FALSE;
	END_IF
	
// Gripper is moved down to grab the piece
043:
	moveTest.zPos := zDown;
	caseState := 044;
	
// Move is executed
044:
	moveTest.ExecuteMove := TRUE;
	caseState := 046;

// Gripper is in position to pick up jumped piece
// Gripper is closed around the piece that is to be jumped
046:
	IF(moveTest.MoveDone)THEN
		caseState := 047;
		moveTest.ExecuteMove := FALSE;
		GripperMove := TRUE;
		wait.startTimer := TRUE;
	END_IF

// Gripper will be moved up
047:
	IF(wait.done) THEN
		wait.startTimer := FALSE;
		moveTest.zPos := zUp;
		caseState := 048;
	END_IF
	
// Move is executed
048: 
	moveTest.ExecuteMove := TRUE;
	caseState := 049;

// Move is completed
// At this point, the piece is grabbed and ready discarded to its correct stack
049:
	IF(moveTest.MoveDone)THEN
		caseState := 050;
		moveTest.ExecuteMove := FALSE;
	END_IF
	
// Moves above stack where piece is to be dropped off
// Calculated based on color and current stack, etc.
050:	
	// update all stack information so that the next piece will be dropped off correctly
	IF(redOrBlack = 0) THEN // jumping piece is red, so jumped piece is black (add to the black stack)
		moveTest.xPos := blackStackXOffset + (GVL.currentBlackStack * stackXDistApart);
		moveTest.yPos := blackStackYOffset + (GVL.currentBlackStack * stackYDistApart);		
	ELSE // jumping piece is black, so jumped piece is red (add to the red stack)
		moveTest.xPos := redStackXOffset + (GVL.currentRedStack * stackXDistApart);
		moveTest.yPos := redStackYOffset + (GVL.currentRedStack * stackYDistApart);	
	END_IF
	moveTest.zPos := zUp;		
	jumpCounter := jumpCounter + 1;
	caseState := 051;




	
	
	
// Move is executed
051:
	moveTest.ExecuteMove := TRUE;
	caseState := 052;
	
// Move is complete
052:
	IF(moveTest.MoveDone) THEN
		caseState := 053;
		moveTest.ExecuteMove := FALSE;
	END_IF
	
// Calculates where piece should be placed in the current stack
// Updates the position in the stack so it points to the NEXT AVAILABLE spot in the stack
// Stack position counts up from the bottom, with the bottom-most position being position 0 
// and the top-most position being position 4
053:
	IF(redOrBlack = 0) THEN // jumping piece is red, so jumped piece is black (add to the black stack)
		moveTest.zPos := zDown - ((4 - GVL.currentBlackStackPos) * pieceOffset);
		GVL.currentBlackStackPos := GVL.currentBlackStackPos - 1;
		IF(GVL.currentBlackStackPos < 0) THEN
			GVL.currentBlackStackPos := 4;
			GVL.currentBlackStack := GVL.currentBlackStack - 1;
		END_IF
	ELSE
		moveTest.zPos := zDown - ((4 - GVL.currentRedStackPos) * pieceOffset);
		GVL.currentRedStackPos := GVL.currentRedStackPos - 1;
		IF(GVL.currentRedStackPos < 0) THEN
			GVL.currentRedStackPos := 4;
			GVL.currentRedStack := GVL.currentRedStack - 1;
		END_IF
	END_IF
	caseState := 054;

// Move is executed
054:
	moveTest.ExecuteMove := TRUE;
	caseState := 055;

// Piece is dropped off in the appropriate stack position
055:
	IF(moveTest.MoveDone)THEN
		caseState := 056;
		moveTest.ExecuteMove := FALSE;
		GripperMove := FALSE;
		wait.startTimer := TRUE;
	END_IF

// Gripper is done with its wait, the up position is commanded
056:
	IF(wait.done)THEN
		wait.startTimer := FALSE;
		moveTest.zPos := zUp;
		caseState := 057;
	END_IF
	
// Move is executed
057:
	moveTest.ExecuteMove := TRUE;
	caseState := 058;

// Move to up position is complete
058:
	IF(moveTest.MoveDone) THEN
		caseState := 040;
		moveTest.ExecuteMove := FALSE;
	END_IF

// After all jumped pieces have been removed, kinging will take place
// kingCurrentPiece is set to true if a piece achieves king status in a given turn
// Only one piece can be kinged per turn
070:
	IF(kingCurrentPiece AND redOrBlack = 0)THEN // current piece has achieved king status and is red
		// Because the current stack position points to the NEXT OPEN stack space
		// the current stack position needs to be decremented so it points to the first ACTUAL PIECE
		GVL.currentRedStackPos := GVL.currentRedStackPos + 1;
		IF(GVL.currentRedStackPos > 4)THEN
			GVL.currentRedStack := GVL.currentRedStack + 1;
			GVL.currentRedStackPos := 0;
		END_IF	
		IF(GVL.currentRedStack > 2) THEN // this would mean there is no piece that can be used for kinging
			caseState := 100;
		ELSE
			moveTest.xPos := redStackXOffset + (GVL.currentRedStack * stackXDistApart);
			moveTest.yPos := redStackYOffset + (GVL.currentRedStack * stackYDistApart);
			moveTest.zPos := zUp;
			caseState := 071;
		END_IF

	ELSIF(kingCurrentPiece AND redOrBlack = 1) THEN // current piece has achieved king status and is black
		GVL.currentBlackStackPos := GVL.currentBlackStackPos + 1;
		IF(GVL.currentBlackStackPos > 4)THEN
			GVL.currentBlackStack := GVL.currentBlackStack + 1;
		END_IF	
		IF(GVL.currentBlackStack > 2) THEN // this would mean there is no piece that can be used for kinging
			caseState := 100;
		ELSE
			moveTest.xPos := blackStackXOffset + (GVL.currentBlackStack * stackXDistApart);
			moveTest.yPos := blackStackYOffset + (GVL.currentBlackStack * stackYDistApart);	
			moveTest.zPos := zUp;
			caseState := 071;
		END_IF
	ELSE // no piece achieved king status on that turn, end the turn
		caseState := 100;
END_IF

// Move is executed	
071:
	moveTest.ExecuteMove := TRUE;
	caseState := 072;

// Gripper is now above the stack where the piece will be taken to be added to the king
072:
	IF(moveTest.MoveDone) THEN
		caseState := 073;
		moveTest.ExecuteMove := FALSE;
	END_IF

// This case cannot be reached unless a piece has achieved king status on this turn
// Sets position to where the piece needs to be picked up based on current stack position
073:
	IF(redOrBlack = 0) THEN // kinged piece is red and going to grab a red piece
		moveTest.zPos := zDown - ((4 - GVL.currentRedStackPos) * pieceOffset);
	ELSE // kinged piece is black
		moveTest.zPos := zDown - ((4 - GVL.currentBlackStackPos) * pieceOffset);
	END_IF
	caseState := 074;

// Move is executed
074:
	moveTest.ExecuteMove := TRUE;
	caseState := 075;

// Grab piece to be used as the kinging piece
075:
	IF(moveTest.MoveDone)THEN
		caseState := 076;
		moveTest.ExecuteMove := FALSE;
		GripperMove := TRUE;
		wait.startTimer := TRUE;
	END_IF

// Piece is grabbed and gripper is set to be moved upward
076:
	IF(wait.done)THEN
		wait.startTimer := FALSE;
		moveTest.zPos := zUp;
		caseState := 0765;
	END_IF

// Move is executed	
0765:
	moveTest.ExecuteMove := TRUE;
	caseState := 0766;

// Move is done
0766:
	IF(moveTest.MoveDone)THEN
		caseState := 077;
		moveTest.ExecuteMove := FALSE;
	END_IF

// Gripper is positioned over the piece to be kinged; the second piece is currently held in the gripper
077:
	moveTest.xPos := xOffset + (currentPiece.currentLocation[0] * spaceOffset);
	moveTest.yPos := yOffset + (currentPiece.currentLocation[1] * spaceOffset);
	moveTest.zPos := zUp;
	caseState := 078;

// Move is executed
078:
	moveTest.ExecuteMove := TRUE;
	caseState := 079;

// Move is completed
079:
	IF(moveTest.MoveDone)THEN
		caseState := 080;
		moveTest.ExecuteMove := FALSE;
	END_IF

// Z position is set to 1 piece-height above the board and directly over the kinged piece
080:
	moveTest.zPos := zDown - pieceOffset;
	caseState := 081;

// Move is executed
081:
	moveTest.ExecuteMove := TRUE;
	caseState := 082;

// Drops piece on piece to be kinged
082:
	IF(moveTest.MoveDone)THEN
		caseState := 083;
		moveTest.ExecuteMove := FALSE;
		GripperMove := FALSE;
		wait.startTimer := TRUE;
	END_IF

// Commanded move is straight up	
083: 
	IF(wait.done)THEN
		wait.startTimer := FALSE;
		moveTest.zPos := zUp;
		caseState := 084;
	END_IF

// Move is executed
084:
	moveTest.ExecuteMove := TRUE;
	caseState := 085;

// Move is complete
// King current piece is set to false so it will not be run next time
// (Unless a piece achieves king status next time)
085:
	IF(moveTest.MoveDone) THEN
		caseState := 100;
		moveTest.ExecuteMove := FALSE;
		kingCurrentPiece := FALSE;
	END_IF
	
// ALL OPERATIONS HAVE BEEN COMPLETED
// CASE is set to 000, and the entire operation will be executed next turn	
// There is a check to see if a player has won
100:
	IF(NOT moveTest.ExecuteMove) THEN
		IF(GVL.redWins OR GVL.blackWins)THEN
			caseState := 200;
		ELSE
			caseState := 000;
		END_IF
		
	END_IF
	

END_CASE

// THESE CALLS WILL RUN EVERY BUS CYCLE
// THEIR EXECUTE IS CONTROLLED BY ALL OF THE CASE STATEMENTS IN THE ABOVE CODE
moveTest();
wait();

END_PROGRAM

// CODESYS_SoftMotion_Win_V3/Application/GameplayFunctions/findSelectedPiece
FUNCTION findSelectedPiece : ARRAY [0..1] OF INT
VAR_INPUT
END_VAR
VAR
	i : INT;
END_VAR

FOR i := 0 TO 11 DO
	IF(GVL.pieces[0,i].isSelected) THEN
		findSelectedPiece[0] := 0;
		findSelectedPiece[1] := i;
	END_IF
	IF(GVL.pieces[1,i].isSelected) THEN
		findSelectedPiece[0] := 1;
		findSelectedPiece[1] := i;
	END_IF
END_FOR

RETURN;

END_FUNCTION

// CODESYS_SoftMotion_Win_V3/Application/GameplayFunctions/MakeJump
PROGRAM MakeJump
VAR
	pieceColor : INT;
	pieceIndex : INT;
	
	jumpedColor : INT;
	jumpedIndex : INT;
	
	jumpedLocX : INT := -1;
	jumpedLocY : INT := -1;
	
	temp : ARRAY [0..1] OF INT;
	
	i : INT;
	j : INT := 0;
	
	usedJumpProfile : INT;
	lengthJumpSeq : INT := -1;
END_VAR

// Null out global variables that are used when taking pieces that are jumped
GVL.takenList := GVL.emptyTakenList;
GVL.takenListLength := 0;
lengthJumpSeq := -1;

// Finds the index of the selected piece that is making a move
temp := findSelectedPiece();
pieceColor := temp[0];
pieceIndex := temp[1];

// Finds longest jump profile that ends at the chosen destination space
FOR i := 20 TO 0 BY -1 DO 
	
	j := 0;
	WHILE(j < 4 AND GVL.pieces[pieceColor, pieceIndex].jumpArr[i,j].xMoveLocation <> -1) DO
		IF(GVL.pieces[pieceColor, pieceIndex].jumpArr[i,j].xMoveLocation = GVL.xMoveSpace AND GVL.pieces[pieceColor, pieceIndex].jumpArr[i,j].yMoveLocation = GVL.yMoveSpace AND j > lengthJumpSeq)THEN
			usedJumpProfile := i;
			lengthJumpSeq := j;
		END_IF
		j := j + 1;
	END_WHILE

END_FOR

GVL.takenListLength := lengthJumpSeq + 1;

FOR i := 0 TO lengthJumpSeq DO
	// assigns easy to read values to piece that is to be jumped
	jumpedColor := GVL.pieces[pieceColor, pieceIndex].jumpArr[usedJumpProfile,i].jumpedColor;
	jumpedIndex := GVL.pieces[pieceColor, pieceIndex].jumpArr[usedJumpProfile,i].jumpedIndex;
	IF(jumpedColor >= 0) THEN
		jumpedLocX := GVL.pieces[jumpedColor, jumpedIndex].currentLocation[0];
		jumpedLocY := GVL.pieces[jumpedColor, jumpedIndex].currentLocation[1];
		
		GVL.takenList[i,0] := jumpedLocX;
		GVL.takenList[i,1] := jumpedLocY;
	
		GVL.pieces[jumpedColor, jumpedIndex].translatedLocation[0] := 0;
		GVL.pieces[jumpedColor, jumpedIndex].translatedLocation[1] := 0;
	
		// Nulls out information for all taken pieces
		GVL.pieces[jumpedColor, jumpedIndex].isTaken := TRUE;
		GVL.pieces[jumpedColor, jumpedIndex].isKing := FALSE;
	
		// Makes location an invalid value
		GVL.pieces[jumpedColor, jumpedIndex].currentLocation[0] := -1;
		GVL.pieces[jumpedColor, jumpedIndex].currentLocation[1] := -1;
	
		// Makes the taken piece have zero valid moves
		GVL.pieces[jumpedColor, jumpedIndex].validMoveArr := GVL.noValidMoveArr;
	
		WHILE(jumpedLocX = 0 AND jumpedLocY = 0) DO
			//
		END_WHILE
	
		// Clears board space that was occupied by the taken piece
		GVL.board[jumpedLocX, jumpedLocY].isEmpty := TRUE;
		GVL.board[jumpedLocX, jumpedLocY].isRed := FALSE;
		GVL.board[jumpedLocX, jumpedLocY].isBlack := FALSE;
	END_IF			
END_FOR

END_PROGRAM

// CODESYS_SoftMotion_Win_V3/Application/GameplayFunctions/UpdateValidMoveArrays
PROGRAM UpdateValidMoveArrays
VAR
	i : INT;
	x: INT;
	y : INT;
	xNext : INT;
	yNext : INT;
END_VAR

// Code will run continuously, but will not execute until board is setup
// If code runs before board is setup, there will be an error, so don't do that ok?
IF(GVL.boardIsSetup)THEN	
	// Checks moves for red
	IF(GVL.redsTurn) THEN
	GVL.currentJumpRef := 0;
	FOR i:= 0 TO 11 DO
		GVL.pieces[0,i].validMoveArr := GVL.noValidMoveArr;
		x:= GVL.pieces[0,i].currentLocation[0];
		y := GVL.pieces[0,i].currentLocation[1];
	
		// Checks for move up and right
		IF(x+1 < 8 AND y+1 < 8 AND GVL.board[x+1,y+1].isEmpty) THEN
			GVL.pieces[0,i].validMoveArr[x+1,y+1] := TRUE;
		END_IF

		// Checks for move up and left
		IF(x-1 >= 0 AND y+1 < 8 AND GVL.board[x-1,y+1].isEmpty) THEN
			GVL.pieces[0,i].validMoveArr[x-1,y+1] := TRUE;
		END_IF
		
		// Checks for move down and left (FOR KINGS ONLY)
		IF(x-1 >= 0 AND y-1 >= 0 AND GVL.board[x-1,y-1].isEmpty AND GVL.pieces[0,i].isKing) THEN
			GVL.pieces[0,i].validMoveArr[x-1,y-1] := TRUE;
		END_IF
		
		// Checks for move down and right (FOR KINGS ONLY)
		IF(x+1 >= 0 AND y-1 >= 0 AND GVL.board[x+1,y-1].isEmpty AND GVL.pieces[0,i].isKing) THEN
			GVL.pieces[0,i].validMoveArr[x+1,y-1] := TRUE;
		END_IF
		
		// Checks for all red jumps (pseudo recursive call)
		clearGlobalStack();
		GVL.currentStackIndex := 0;
		GVL.currentJumpProfileNum := 0;
		clearPieceJumpArray(0,i);
		GVL.pieces[0,i] := checkForJumpRed1(GVL.pieces[0,i], i);
		
	END_FOR
	
	ELSE
	GVL.currentJumpRef := 0;
	// Setup valid moves for black
	FOR i:= 0 TO 11 DO
		GVL.pieces[1,i].validMoveArr := GVL.noValidMoveArr;
		x:= GVL.pieces[1,i].currentLocation[0];
		y := GVL.pieces[1,i].currentLocation[1];
	
		// Checks for down and right
		IF(x+1 < 8 AND y-1 >= 0 AND GVL.board[x+1,y-1].isEmpty) THEN
			GVL.pieces[1,i].validMoveArr[x+1,y-1] := TRUE;
		END_IF

		// Checks for move down and left
		IF(x-1 >= 0 AND y-1 >= 0 AND GVL.board[x-1,y-1].isEmpty) THEN
			GVL.pieces[1,i].validMoveArr[x-1,y-1] := TRUE;
		END_IF
		
		// Checks for move up and left (FOR KINGS ONLY)
		IF(x-1 >= 0 AND y+1 >= 0 AND GVL.board[x-1,y+1].isEmpty AND GVL.pieces[1,i].isKing) THEN
			GVL.pieces[1,i].validMoveArr[x-1,y+1] := TRUE;
		END_IF
		
		// Checks for move up and right (FOR KINGS ONLY)
		IF(x+1 >= 0 AND y+1 >= 0 AND GVL.board[x+1,y+1].isEmpty AND GVL.pieces[1,i].isKing) THEN
			GVL.pieces[1,i].validMoveArr[x+1,y+1] := TRUE;
		END_IF
	
		clearGlobalStack();
		GVL.currentStackIndex := 0;
		GVL.currentJumpProfileNum := 0;
		clearPieceJumpArray(0,i);
		GVL.pieces[1,i] := checkForJumpBlack1(GVL.pieces[1,i], i);
		(*
		IF(x+1 < 8 AND y+1 < 8 AND NOT GVL.board[x+1,y+1].isEmpty AND GVL.board[x+1,y+1].isBlack) THEN
		
			//possible jump
		END_IF
		*)
		
	END_FOR
	END_IF
END_IF

END_PROGRAM

// CODESYS_SoftMotion_Win_V3/Application/GameplayFunctions/clearGlobalStack
FUNCTION clearGlobalStack : bool
VAR_INPUT
END_VAR
VAR
	i : INT := 0;
END_VAR

FOR i := 0 TO 3 DO
	GVL.jumpStack[i].jumpedColor := -1;
	GVL.jumpStack[i].jumpedIndex:= -1;
	GVL.jumpStack[i].xMoveLocation := -1;
	GVL.jumpStack[i].yMoveLocation := -1;
END_FOR

END_FUNCTION

// CODESYS_SoftMotion_Win_V3/Application/GameplayFunctions/clearPieceJumpArray
FUNCTION clearPieceJumpArray : BOOL
VAR_INPUT
	pieceColor : INT;
	pieceIndex : INT;
END_VAR
VAR
	i : INT;
END_VAR

FOR i := 0 TO 11 DO
	GVL.pieces[pieceColor,pieceIndex].jumpArr := GVL.emptyJumpArr;
END_FOR

END_FUNCTION

// CODESYS_SoftMotion_Win_V3/Application/GameplayFunctions/checkForJumpRed1
FUNCTION checkForJumpRed1 : Piece
VAR_INPUT
	selectedPiece : Piece;
	selectedPieceIndex : INT;
END_VAR

VAR
	i : INT;
	x: INT;
	y: INT;
	xNext : INT;
	yNext : INT;
	jumpedPieceIndex : INT;
	temp : ARRAY [0..1] OF INT;
END_VAR

x := selectedPiece.currentLocation[0];
y := selectedPiece.currentLocation[1];

// checks the board space up and to the right
IF(x+1 < 8 AND y+1 < 8 AND NOT GVL.board[x+1,y+1].isEmpty AND GVL.board[x+1,y+1].isBlack) THEN
	xNext := x + 2; // location of the space you could possibly jump to
	yNext := y + 2; // location of the space you could possibly jump to		
	// if the space that can be jumped to is 
	IF(xNext < 8 AND yNext < 8 AND GVL.board[xNext,yNext].isEmpty) THEN
		selectedPiece.validMoveArr[xNext,yNext] := TRUE;
		temp := findPieceAtGivenLocation(x+1,y+1);
		jumpedPieceIndex := temp[1];
		IF(push(1, jumpedPieceIndex, xNext, yNext)) THEN
			selectedPiece := checkForJumpRed2(selectedPiece, selectedPieceIndex, xNext, yNext);
			selectedPiece := pop(selectedPiece, 0);
		END_IF
	END_IF
END_IF

// checks up and to the left
IF(x-1 >= 0 AND y+1 < 8 AND NOT GVL.board[x-1,y+1].isEmpty AND GVL.board[x-1,y+1].isBlack) THEN
	xNext := x - 2; // location of the space you could possibly jump to
	yNext := y + 2; // location of the space you could possibly jump to
	IF(xNext >= 0 AND yNext < 8 AND GVL.board[xNext,yNext].isEmpty) THEN
		selectedPiece.validMoveArr[xNext,yNext] := TRUE;
		temp := findPieceAtGivenLocation(x-1,y+1);
		jumpedPieceIndex := temp[1];
		IF(push(1, jumpedPieceIndex, xNext, yNext)) THEN
			selectedPiece := checkForJumpRed2(selectedPiece, selectedPieceIndex, xNext, yNext);
			selectedPiece := pop(selectedPiece, 0);
		END_IF
	END_IF
END_IF

// checks down and left
IF(x-1 >= 0 AND y-1 < 8 AND NOT GVL.board[x-1,y-1].isEmpty AND GVL.board[x-1,y-1].isBlack AND selectedPiece.isKing) THEN
	xNext := x - 2; // location of the space you could possibly jump to
	yNext := y - 2; // location of the space you could possibly jump to
	IF(xNext >= 0 AND yNext < 8 AND GVL.board[xNext,yNext].isEmpty) THEN
		selectedPiece.validMoveArr[xNext,yNext] := TRUE;
		temp := findPieceAtGivenLocation(x-1,y-1);
		jumpedPieceIndex := temp[1];
		IF(push(1, jumpedPieceIndex, xNext, yNext)) THEN
			selectedPiece := checkForJumpRed2(selectedPiece, selectedPieceIndex, xNext, yNext);
			selectedPiece := pop(selectedPiece, 0);
		END_IF
	END_IF
END_IF

// checks down and right
IF(x+1 >= 0 AND y-1 < 8 AND NOT GVL.board[x+1,y-1].isEmpty AND GVL.board[x+1,y-1].isBlack AND selectedPiece.isKing) THEN
	xNext := x + 2; // location of the space you could possibly jump to
	yNext := y - 2; // location of the space you could possibly jump to
	IF(xNext >= 0 AND yNext < 8 AND GVL.board[xNext,yNext].isEmpty) THEN
		selectedPiece.validMoveArr[xNext,yNext] := TRUE;
		temp := findPieceAtGivenLocation(x+1,y-1);
		jumpedPieceIndex := temp[1];
		IF(push(1, jumpedPieceIndex, xNext, yNext)) THEN
			selectedPiece := checkForJumpRed2(selectedPiece, selectedPieceIndex, xNext, yNext);
			selectedPiece := pop(selectedPiece, 0);
		END_IF
	END_IF
END_IF

checkForJumpRed1 := selectedPiece;


RETURN;

END_FUNCTION

// CODESYS_SoftMotion_Win_V3/Application/GameplayFunctions/findPieceAtGivenLocation
FUNCTION findPieceAtGivenLocation : ARRAY[0..1] OF INT
VAR_INPUT
	xLoc : INT;
	yLoc : INT;
END_VAR
VAR
	i : INT;
END_VAR

FOR i := 0 TO 11 DO
	IF(GVL.pieces[0,i].currentLocation[0] = xLoc AND GVL.pieces[0,i].currentLocation[1] = yLoc) THEN
		findPieceAtGivenLocation[0] := 0;
		findPieceAtGivenLocation[1] := i;
	END_IF
	IF(GVL.pieces[1,i].currentLocation[0] = xLoc AND GVL.pieces[1,i].currentLocation[1] = yLoc) THEN
		findPieceAtGivenLocation[0] := 1;
		findPieceAtGivenLocation[1] := i;
	END_IF
END_FOR
RETURN;

END_FUNCTION

// CODESYS_SoftMotion_Win_V3/Application/GameplayFunctions/push
FUNCTION push : bool
VAR_INPUT
	jumpedColor : INT;
	jumpedIndex : INT;
	xMoveLoc : INT;
	yMoveLoc : INT;
END_VAR
VAR
	
END_VAR

IF(GVL.currentStackIndex < 4) THEN
	
	// Adds jump information to the current stack
	GVL.jumpStack[GVL.currentStackIndex].xMoveLocation := xMoveLoc;
	GVL.jumpStack[GVL.currentStackIndex].yMoveLocation := yMoveLoc;
	GVL.jumpStack[GVL.currentStackIndex].jumpedColor := jumpedColor;
	GVL.jumpStack[GVL.currentStackIndex].jumpedIndex := jumpedIndex;
	
	// Moves top of the stack up one notch
	GVL.currentStackIndex := GVL.currentStackIndex + 1;
	
	push := TRUE;
ELSE
	// Would indicate that the stack is full (only 4 successive jumps are allowed)
	push := FALSE;
END_IF

END_FUNCTION

// CODESYS_SoftMotion_Win_V3/Application/GameplayFunctions/checkForJumpRed2
FUNCTION checkForJumpRed2 : Piece
VAR_INPUT
	selectedPiece : Piece;
	selectedPieceIndex : INT;
	x : INT;
	y : INT;
END_VAR


VAR
	jumpedPieceIndex : INT;
	xNext : INT;
	yNext : INT;
	i : INT;
	temp: ARRAY [0..1] OF INT;
END_VAR

// checks up and to the right
IF(x+1 < 8 AND y+1 < 8 AND NOT GVL.board[x+1,y+1].isEmpty AND GVL.board[x+1,y+1].isBlack) THEN
	xNext := x + 2; // location of the space you could possibly jump to
	yNext := y + 2; // location of the space you could possibly jump to		
	temp := findPieceAtGivenLocation(x+1,y+1);
	selectedPieceIndex := temp[1];
	IF(xNext < 8 AND yNext < 8 AND GVL.board[xNext,yNext].isEmpty) THEN
		selectedPiece.validMoveArr[xNext,yNext] := TRUE;	
		temp := findPieceAtGivenLocation(x+1,y+1);
		jumpedPieceIndex := temp[1];
		IF(push(1, jumpedPieceIndex, xNext, yNext))THEN
			selectedPiece := checkForJumpRed3(selectedPiece, selectedPieceIndex, xNext, yNext);	
			selectedPiece := pop(selectedPiece, 0);
		END_IF
	END_IF
END_IF

// checks up and to the left
IF(x-1 >= 0 AND y+1 < 8 AND NOT GVL.board[x-1,y+1].isEmpty AND GVL.board[x-1,y+1].isBlack) THEN
	xNext := x - 2; // location of the space you could possibly jump to
	yNext := y + 2; // location of the space you could possibly jump to
	IF(xNext >= 0 AND yNext < 8 AND GVL.board[xNext,yNext].isEmpty) THEN
		selectedPiece.validMoveArr[xNext,yNext] := TRUE;
		temp := findPieceAtGivenLocation(x-1,y+1);
		jumpedPieceIndex := temp[1];
		IF(push(1, jumpedPieceIndex, xNext, yNext))THEN
			selectedPiece := checkForJumpRed3(selectedPiece, selectedPieceIndex, xNext, yNext);	
			selectedPiece := pop(selectedPiece, 0);
		END_IF
	END_IF
END_IF

// checks down and left
IF(x-1 >= 0 AND y-1 < 8 AND NOT GVL.board[x-1,y-1].isEmpty AND GVL.board[x-1,y-1].isBlack AND selectedPiece.isKing) THEN
	xNext := x - 2; // location of the space you could possibly jump to
	yNext := y - 2; // location of the space you could possibly jump to
	IF(xNext >= 0 AND yNext < 8 AND GVL.board[xNext,yNext].isEmpty) THEN
		selectedPiece.validMoveArr[xNext,yNext] := TRUE;
		temp := findPieceAtGivenLocation(x-1,y-1);
		jumpedPieceIndex := temp[1];
		IF(push(1, jumpedPieceIndex, xNext, yNext)) THEN
			selectedPiece := checkForJumpRed3(selectedPiece, selectedPieceIndex, xNext, yNext);
			selectedPiece := pop(selectedPiece, 0);
		END_IF
	END_IF
END_IF

// checks down and right
IF(x+1 >= 0 AND y-1 < 8 AND NOT GVL.board[x+1,y-1].isEmpty AND GVL.board[x+1,y-1].isBlack AND selectedPiece.isKing) THEN
	xNext := x + 2; // location of the space you could possibly jump to
	yNext := y - 2; // location of the space you could possibly jump to
	IF(xNext >= 0 AND yNext < 8 AND GVL.board[xNext,yNext].isEmpty) THEN
		selectedPiece.validMoveArr[xNext,yNext] := TRUE;
		temp := findPieceAtGivenLocation(x+1,y-1);
		jumpedPieceIndex := temp[1];
		IF(push(1, jumpedPieceIndex, xNext, yNext)) THEN
			selectedPiece := checkForJumpRed3(selectedPiece, selectedPieceIndex, xNext, yNext);
			selectedPiece := pop(selectedPiece, 0);
		END_IF
	END_IF
END_IF

checkForJumpRed2 := selectedPiece;


RETURN;

END_FUNCTION

// CODESYS_SoftMotion_Win_V3/Application/GameplayFunctions/checkForJumpRed3
FUNCTION checkForJumpRed3 : Piece
VAR_INPUT
	selectedPiece : Piece;
	selectedPieceIndex : INT;
	x : INT;
	y : INT; 
END_VAR

VAR
	xNext : INT;
	yNext : INT;
	i :INT;
	temp: ARRAY [0..1] OF INT;
	jumpedPieceIndex: INT;
END_VAR

// checks up and to the right
IF(x+1 < 8 AND y+1 < 8 AND NOT GVL.board[x+1,y+1].isEmpty AND GVL.board[x+1,y+1].isBlack) THEN
	xNext := x + 2; // location of the space you could possibly jump to
	yNext := y + 2; // location of the space you could possibly jump to		

	IF(xNext < 8 AND yNext < 8 AND GVL.board[xNext,yNext].isEmpty) THEN
		selectedPiece.validMoveArr[xNext,yNext] := TRUE;
		temp := findPieceAtGivenLocation(x+1,y+1);
		jumpedPieceIndex := temp[1];
		IF(push(1, jumpedPieceIndex, xNext, yNext))THEN
			selectedPiece := checkForJumpRed4(selectedPiece, selectedPieceIndex, xNext, yNext);	
			selectedPiece := pop(selectedPiece, 0);
		END_IF
	END_IF
END_IF

// checks up and to the left
IF(x-1 >= 0 AND y+1 < 8 AND NOT GVL.board[x-1,y+1].isEmpty AND GVL.board[x-1,y+1].isBlack) THEN
	xNext := x - 2; // location of the space you could possibly jump to
	yNext := y + 2; // location of the space you could possibly jump to
	IF(xNext >= 0 AND yNext < 8 AND GVL.board[xNext,yNext].isEmpty) THEN
		selectedPiece.validMoveArr[xNext,yNext] := TRUE;
		temp := findPieceAtGivenLocation(x-1,y+1);
		jumpedPieceIndex := temp[1];
		IF(push(1, jumpedPieceIndex, xNext, yNext))THEN
			selectedPiece := checkForJumpRed4(selectedPiece, selectedPieceIndex, xNext, yNext);	
			selectedPiece := pop(selectedPiece, 0);
		END_IF
	END_IF
END_IF

// checks down and left
IF(x-1 >= 0 AND y-1 < 8 AND NOT GVL.board[x-1,y-1].isEmpty AND GVL.board[x-1,y-1].isBlack AND selectedPiece.isKing) THEN
	xNext := x - 2; // location of the space you could possibly jump to
	yNext := y - 2; // location of the space you could possibly jump to
	IF(xNext >= 0 AND yNext < 8 AND GVL.board[xNext,yNext].isEmpty) THEN
		selectedPiece.validMoveArr[xNext,yNext] := TRUE;
		temp := findPieceAtGivenLocation(x-1,y-1);
		jumpedPieceIndex := temp[1];
		IF(push(1, jumpedPieceIndex, xNext, yNext)) THEN
			selectedPiece := checkForJumpRed4(selectedPiece, selectedPieceIndex, xNext, yNext);
			selectedPiece := pop(selectedPiece, 0);
		END_IF
	END_IF
END_IF

// checks down and right
IF(x+1 >= 0 AND y-1 < 8 AND NOT GVL.board[x+1,y-1].isEmpty AND GVL.board[x+1,y-1].isBlack AND selectedPiece.isKing) THEN
	xNext := x + 2; // location of the space you could possibly jump to
	yNext := y - 2; // location of the space you could possibly jump to
	IF(xNext >= 0 AND yNext < 8 AND GVL.board[xNext,yNext].isEmpty) THEN
		selectedPiece.validMoveArr[xNext,yNext] := TRUE;
		temp := findPieceAtGivenLocation(x+1,y-1);
		jumpedPieceIndex := temp[1];
		IF(push(1, jumpedPieceIndex, xNext, yNext)) THEN
			selectedPiece := checkForJumpRed4(selectedPiece, selectedPieceIndex, xNext, yNext);
			selectedPiece := pop(selectedPiece, 0);
		END_IF
	END_IF
END_IF

checkForJumpRed3 := selectedPiece;


RETURN;

END_FUNCTION

// CODESYS_SoftMotion_Win_V3/Application/GameplayFunctions/checkForJumpRed4
FUNCTION checkForJumpRed4 : Piece
VAR_INPUT
	selectedPiece : Piece;
	selectedPieceIndex: INT;
	x : INT;
	y : INT; 
END_VAR

VAR
	xNext : INT;
	yNext : INT;
	temp: ARRAY [0..1] OF INT;
	jumpedPieceIndex: INT;
	
END_VAR

// checks up and to the right
IF(x+1 < 8 AND y+1 < 8 AND NOT GVL.board[x+1,y+1].isEmpty AND GVL.board[x+1,y+1].isBlack) THEN
	xNext := x + 2; // location of the space you could possibly jump to
	yNext := y + 2; // location of the space you could possibly jump to		
	IF(xNext < 8 AND yNext < 8 AND GVL.board[xNext,yNext].isEmpty) THEN
		selectedPiece.validMoveArr[xNext,yNext] := TRUE;
		temp := findPieceAtGivenLocation(x+1,y+1);
		jumpedPieceIndex := temp[1];
		IF(push(1, jumpedPieceIndex, xNext, yNext))THEN
			// This is where another jump would be called	
			selectedPiece := pop(selectedPiece, 0);
		END_IF		
	END_IF
END_IF

// checks up and to the left
IF(x-1 >= 0 AND y+1 < 8 AND NOT GVL.board[x-1,y+1].isEmpty AND GVL.board[x-1,y+1].isBlack) THEN
	xNext := x - 2; // location of the space you could possibly jump to
	yNext := y + 2; // location of the space you could possibly jump to
	IF(xNext >= 0 AND yNext < 8 AND GVL.board[xNext,yNext].isEmpty) THEN
		selectedPiece.validMoveArr[xNext,yNext] := TRUE;
		temp := findPieceAtGivenLocation(x-1,y+1);
		jumpedPieceIndex := temp[1];
		IF(push(1, jumpedPieceIndex, xNext, yNext))THEN
			// This is where you would call another jump
			selectedPiece := pop(selectedPiece, 0);
		END_IF	
	
	END_IF
END_IF

// checks down and left (KINGS ONLY)
IF(x-1 >= 0 AND y-1 < 8 AND NOT GVL.board[x-1,y-1].isEmpty AND GVL.board[x-1,y-1].isBlack AND selectedPiece.isKing) THEN
	xNext := x - 2; // location of the space you could possibly jump to
	yNext := y - 2; // location of the space you could possibly jump to
	IF(xNext >= 0 AND yNext < 8 AND GVL.board[xNext,yNext].isEmpty) THEN
		selectedPiece.validMoveArr[xNext,yNext] := TRUE;
		temp := findPieceAtGivenLocation(x-1,y-1);
		jumpedPieceIndex := temp[1];
		IF(push(1, jumpedPieceIndex, xNext, yNext)) THEN
			//selectedPiece := checkForJumpRed2(selectedPiece, selectedPieceIndex, xNext, yNext);
			selectedPiece := pop(selectedPiece, 0);
		END_IF
	END_IF
END_IF

// checks down and right (KINGS ONLY)
IF(x+1 >= 0 AND y-1 < 8 AND NOT GVL.board[x+1,y-1].isEmpty AND GVL.board[x+1,y-1].isBlack AND selectedPiece.isKing) THEN
	xNext := x + 2; // location of the space you could possibly jump to
	yNext := y - 2; // location of the space you could possibly jump to
	IF(xNext >= 0 AND yNext < 8 AND GVL.board[xNext,yNext].isEmpty) THEN
		selectedPiece.validMoveArr[xNext,yNext] := TRUE;
		temp := findPieceAtGivenLocation(x+1,y-1);
		jumpedPieceIndex := temp[1];
		IF(push(1, jumpedPieceIndex, xNext, yNext)) THEN
			//selectedPiece := checkForJumpRed2(selectedPiece, selectedPieceIndex, xNext, yNext);
			selectedPiece := pop(selectedPiece, 0);
		END_IF
	END_IF
END_IF

checkForJumpRed4 := selectedPiece;


RETURN;

END_FUNCTION

// CODESYS_SoftMotion_Win_V3/Application/GameplayFunctions/pop
FUNCTION pop : Piece
VAR_INPUT
	currentPiece : Piece;
	pieceColor : INT;
END_VAR
VAR
	i : INT := 0;
END_VAR

IF(GVL.currentStackIndex = -1) THEN
	// returns false if stack is empty
	pop := currentPiece;
ELSE
	// save the jumpProfile
	FOR i := 0 TO GVL.currentStackIndex - 1 DO
		currentPiece.jumpArr[GVL.currentJumpProfileNum,i].jumpedColor := GVL.jumpStack[i].jumpedColor;
		currentPiece.jumpArr[GVL.currentJumpProfileNum,i].jumpedIndex := GVL.jumpStack[i].jumpedIndex;
		currentPiece.jumpArr[GVL.currentJumpProfileNum,i].xMoveLocation := GVL.jumpStack[i].xMoveLocation;
		currentPiece.jumpArr[GVL.currentJumpProfileNum,i].yMoveLocation := GVL.jumpStack[i].yMoveLocation;
	END_FOR
	
	GVL.currentJumpProfileNum := GVL.currentJumpProfileNum + 1;
	

	// Pops item off of the stack
	GVL.jumpStack[GVL.currentStackIndex].jumpedColor := -1;
	GVL.jumpStack[GVL.currentStackIndex].jumpedIndex := -1;
	GVL.jumpStack[GVL.currentStackIndex].xMoveLocation := -1;
	GVL.jumpStack[GVL.currentStackIndex].yMoveLocation := -1;
	
	// Moves top of stack down
	GVL.currentStackIndex := GVL.currentStackIndex - 1;
	
	pop := currentPiece;
END_IF

RETURN;

END_FUNCTION

// CODESYS_SoftMotion_Win_V3/Application/GameplayFunctions/checkForJumpBlack1
FUNCTION checkForJumpBlack1 : Piece
VAR_INPUT
	selectedPiece : Piece;
	selectedPieceIndex : INT;
END_VAR

VAR
	x: INT;
	y: INT;
	i : INT;
	xNext : INT;
	yNext : INT;
	temp: ARRAY [0..1] OF INT;
	jumpedPieceIndex: INT;
END_VAR

x := selectedPiece.currentLocation[0];
y := selectedPiece.currentLocation[1];

// checks down and right
IF(x+1 < 8 AND y-1 >= 0 AND NOT GVL.board[x+1,y-1].isEmpty AND GVL.board[x+1,y-1].isRed) THEN
	xNext := x + 2; // location of the space you could possibly jump to
	yNext := y - 2; // location of the space you could possibly jump to		
	IF(xNext < 8 AND yNext >= 0 AND GVL.board[xNext,yNext].isEmpty) THEN
		selectedPiece.validMoveArr[xNext,yNext] := TRUE;
		temp := findPieceAtGivenLocation(x+1,y-1);
		jumpedPieceIndex := temp[1];
		IF(push(0, jumpedPieceIndex, xNext, yNext)) THEN
			selectedPiece := checkForJumpBlack2(selectedPiece, selectedPieceIndex, xNext, yNext);
			selectedPiece := pop(selectedPiece, 1);
		END_IF
	END_IF
END_IF

// checks down and left
IF(x-1 >= 0 AND y-1 >= 0 AND NOT GVL.board[x-1,y-1].isEmpty AND GVL.board[x-1,y-1].isRed) THEN
	xNext := x - 2; // location of the space you could possibly jump to
	yNext := y - 2; // location of the space you could possibly jump to
	IF(xNext >= 0 AND yNext >= 0 AND GVL.board[xNext,yNext].isEmpty) THEN
		selectedPiece.validMoveArr[xNext,yNext] := TRUE;
		temp := findPieceAtGivenLocation(x-1,y-1);
		jumpedPieceIndex := temp[1];
		IF(push(0, jumpedPieceIndex, xNext, yNext)) THEN
			selectedPiece := checkForJumpBlack2(selectedPiece, selectedPieceIndex, xNext, yNext);
			selectedPiece := pop(selectedPiece, 1);
		END_IF
	END_IF
END_IF

// checks up and left (FOR KINGS ONLY)
IF(x-1 < 8 AND y+1 >= 0 AND NOT GVL.board[x-1,y+1].isEmpty AND GVL.board[x-1,y+1].isRed AND selectedPiece.isKing) THEN
	xNext := x - 2; // location of the space you could possibly jump to
	yNext := y + 2; // location of the space you could possibly jump to		
	IF(xNext < 8 AND yNext >= 0 AND GVL.board[xNext,yNext].isEmpty) THEN
		selectedPiece.validMoveArr[xNext,yNext] := TRUE;
		temp := findPieceAtGivenLocation(x-1,y+1);
		jumpedPieceIndex := temp[1];
		IF(push(0, jumpedPieceIndex, xNext, yNext)) THEN
			selectedPiece := checkForJumpBlack2(selectedPiece, selectedPieceIndex, xNext, yNext);
			selectedPiece := pop(selectedPiece, 1);
		END_IF
	END_IF
END_IF

// checks up and right (FOR KINGS ONLY)
IF(x+1 < 8 AND y+1 >= 0 AND NOT GVL.board[x+1,y+1].isEmpty AND GVL.board[x+1,y+1].isRed AND selectedPiece.isKing) THEN
	xNext := x + 2; // location of the space you could possibly jump to
	yNext := y + 2; // location of the space you could possibly jump to		
	IF(xNext < 8 AND yNext >= 0 AND GVL.board[xNext,yNext].isEmpty) THEN
		selectedPiece.validMoveArr[xNext,yNext] := TRUE;
		temp := findPieceAtGivenLocation(x+1,y+1);
		jumpedPieceIndex := temp[1];
		IF(push(0, jumpedPieceIndex, xNext, yNext)) THEN
			selectedPiece := checkForJumpBlack2(selectedPiece, selectedPieceIndex, xNext, yNext);
			selectedPiece := pop(selectedPiece, 1);
		END_IF
	END_IF
END_IF

checkForJumpBlack1 := selectedPiece;


RETURN;

END_FUNCTION

// CODESYS_SoftMotion_Win_V3/Application/GameplayFunctions/checkForJumpBlack2
FUNCTION checkForJumpBlack2 : Piece
VAR_INPUT
	selectedPiece : Piece;
	selectedPieceIndex : INT;
	x : INT;
	y : INT; 
END_VAR
	
VAR
	i : INT;
	xNext : INT;
	yNext : INT;
	temp: ARRAY [0..1] OF INT;
	jumpedPieceIndex: INT;
END_VAR

// checks down and right
IF(x+1 < 8 AND y-1 >= 0 AND NOT GVL.board[x+1,y-1].isEmpty AND GVL.board[x+1,y-1].isRed) THEN
	xNext := x + 2; // location of the space you could possibly jump to
	yNext := y - 2; // location of the space you could possibly jump to		
	IF(xNext < 8 AND yNext >= 0 AND GVL.board[xNext,yNext].isEmpty) THEN
		selectedPiece.validMoveArr[xNext,yNext] := TRUE;
		temp := findPieceAtGivenLocation(x+1,y-1);
		jumpedPieceIndex := temp[1];
		IF(push(0, jumpedPieceIndex, xNext, yNext)) THEN
			selectedPiece := checkForJumpBlack3(selectedPiece, selectedPieceIndex, xNext, yNext);
			selectedPiece := pop(selectedPiece, 1);
		END_IF
	END_IF
END_IF

// checks down and left
IF(x-1 >= 0 AND y-1 >= 0 AND NOT GVL.board[x-1,y-1].isEmpty AND GVL.board[x-1,y-1].isRed) THEN
	xNext := x - 2; // location of the space you could possibly jump to
	yNext := y - 2; // location of the space you could possibly jump to
	IF(xNext >= 0 AND yNext >= 0 AND GVL.board[xNext,yNext].isEmpty) THEN
		selectedPiece.validMoveArr[xNext,yNext] := TRUE;
		temp := findPieceAtGivenLocation(x-1,y-1);
		jumpedPieceIndex := temp[1];
		IF(push(0, jumpedPieceIndex, xNext, yNext)) THEN
			selectedPiece := checkForJumpBlack3(selectedPiece, selectedPieceIndex, xNext, yNext);
			selectedPiece := pop(selectedPiece, 1);
		END_IF
	END_IF
END_IF

// checks up and left (FOR KINGS ONLY)
IF(x-1 < 8 AND y+1 >= 0 AND NOT GVL.board[x-1,y+1].isEmpty AND GVL.board[x-1,y+1].isRed AND selectedPiece.isKing) THEN
	xNext := x - 2; // location of the space you could possibly jump to
	yNext := y + 2; // location of the space you could possibly jump to		
	IF(xNext < 8 AND yNext >= 0 AND GVL.board[xNext,yNext].isEmpty) THEN
		selectedPiece.validMoveArr[xNext,yNext] := TRUE;
		temp := findPieceAtGivenLocation(x-1,y+1);
		jumpedPieceIndex := temp[1];
		IF(push(0, jumpedPieceIndex, xNext, yNext)) THEN
			selectedPiece := checkForJumpBlack3(selectedPiece, selectedPieceIndex, xNext, yNext);
			selectedPiece := pop(selectedPiece, 1);
		END_IF
	END_IF
END_IF

// checks up and right (FOR KINGS ONLY)
IF(x+1 < 8 AND y+1 >= 0 AND NOT GVL.board[x+1,y+1].isEmpty AND GVL.board[x+1,y+1].isRed AND selectedPiece.isKing) THEN
	xNext := x + 2; // location of the space you could possibly jump to
	yNext := y + 2; // location of the space you could possibly jump to		
	IF(xNext < 8 AND yNext >= 0 AND GVL.board[xNext,yNext].isEmpty) THEN
		selectedPiece.validMoveArr[xNext,yNext] := TRUE;
		temp := findPieceAtGivenLocation(x+1,y+1);
		jumpedPieceIndex := temp[1];
		IF(push(0, jumpedPieceIndex, xNext, yNext)) THEN
			selectedPiece := checkForJumpBlack3(selectedPiece, selectedPieceIndex, xNext, yNext);
			selectedPiece := pop(selectedPiece, 1);
		END_IF
	END_IF
END_IF

checkForJumpBlack2 := selectedPiece;


RETURN;

END_FUNCTION

// CODESYS_SoftMotion_Win_V3/Application/GameplayFunctions/checkForJumpBlack3
FUNCTION checkForJumpBlack3 : Piece
VAR_INPUT
	selectedPiece : Piece;
	selectedPieceIndex : INT;
	x : INT;
	y : INT; 
END_VAR

VAR
	i : INT;
	xNext : INT;
	yNext : INT;
	temp: ARRAY [0..1] OF INT;
	jumpedPieceIndex: INT;
END_VAR

// checks down and right
IF(x+1 < 8 AND y-1 >= 0 AND NOT GVL.board[x+1,y-1].isEmpty AND GVL.board[x+1,y-1].isRed) THEN
	xNext := x + 2; // location of the space you could possibly jump to
	yNext := y - 2; // location of the space you could possibly jump to		
	IF(xNext < 8 AND yNext >= 0 AND GVL.board[xNext,yNext].isEmpty) THEN
		selectedPiece.validMoveArr[xNext,yNext] := TRUE;
		temp := findPieceAtGivenLocation(x+1,y-1);
		jumpedPieceIndex := temp[1];
		IF(push(0, jumpedPieceIndex, xNext, yNext)) THEN
			selectedPiece := checkForJumpBlack4(selectedPiece, selectedPieceIndex, xNext, yNext);
			selectedPiece := pop(selectedPiece, 1);
		END_IF
	END_IF
END_IF

// checks down and left
IF(x-1 >= 0 AND y-1 >= 0 AND NOT GVL.board[x-1,y-1].isEmpty AND GVL.board[x-1,y-1].isRed) THEN
	xNext := x - 2; // location of the space you could possibly jump to
	yNext := y - 2; // location of the space you could possibly jump to
	IF(xNext >= 0 AND yNext >= 0 AND GVL.board[xNext,yNext].isEmpty) THEN
		selectedPiece.validMoveArr[xNext,yNext] := TRUE;
		temp := findPieceAtGivenLocation(x-1,y-1);
		jumpedPieceIndex := temp[1];
		IF(push(0, jumpedPieceIndex, xNext, yNext)) THEN
			selectedPiece := checkForJumpBlack4(selectedPiece, selectedPieceIndex, xNext, yNext);
			selectedPiece := pop(selectedPiece, 1);
		END_IF		
	END_IF
END_IF

// checks up and left (FOR KINGS ONLY)
IF(x-1 < 8 AND y+1 >= 0 AND NOT GVL.board[x-1,y+1].isEmpty AND GVL.board[x-1,y+1].isRed AND selectedPiece.isKing) THEN
	xNext := x - 2; // location of the space you could possibly jump to
	yNext := y + 2; // location of the space you could possibly jump to		
	IF(xNext < 8 AND yNext >= 0 AND GVL.board[xNext,yNext].isEmpty) THEN
		selectedPiece.validMoveArr[xNext,yNext] := TRUE;
		temp := findPieceAtGivenLocation(x-1,y+1);
		jumpedPieceIndex := temp[1];
		IF(push(0, jumpedPieceIndex, xNext, yNext)) THEN
			selectedPiece := checkForJumpBlack4(selectedPiece, selectedPieceIndex, xNext, yNext);
			selectedPiece := pop(selectedPiece, 1);
		END_IF
	END_IF
END_IF

// checks up and right (FOR KINGS ONLY)
IF(x+1 < 8 AND y+1 >= 0 AND NOT GVL.board[x+1,y+1].isEmpty AND GVL.board[x+1,y+1].isRed AND selectedPiece.isKing) THEN
	xNext := x + 2; // location of the space you could possibly jump to
	yNext := y + 2; // location of the space you could possibly jump to		
	IF(xNext < 8 AND yNext >= 0 AND GVL.board[xNext,yNext].isEmpty) THEN
		selectedPiece.validMoveArr[xNext,yNext] := TRUE;
		temp := findPieceAtGivenLocation(x+1,y+1);
		jumpedPieceIndex := temp[1];
		IF(push(0, jumpedPieceIndex, xNext, yNext)) THEN
			selectedPiece := checkForJumpBlack4(selectedPiece, selectedPieceIndex, xNext, yNext);
			selectedPiece := pop(selectedPiece, 1);
		END_IF
	END_IF
END_IF

checkForJumpBlack3 := selectedPiece;


RETURN;

END_FUNCTION

// CODESYS_SoftMotion_Win_V3/Application/GameplayFunctions/checkForJumpBlack4
FUNCTION checkForJumpBlack4 : Piece
VAR_INPUT
	selectedPiece : Piece;
	selectedPieceIndex : INT;
	x : INT;
	y : INT; 
END_VAR

VAR
	xNext : INT;
	yNext : INT;
	temp: ARRAY [0..1] OF INT;
	jumpedPieceIndex: INT;
END_VAR

// checks down and right
IF(x+1 < 8 AND y-1 >= 0 AND NOT GVL.board[x+1,y-1].isEmpty AND GVL.board[x+1,y-1].isRed) THEN
	xNext := x + 2; // location of the space you could possibly jump to
	yNext := y - 2; // location of the space you could possibly jump to		
	IF(xNext < 8 AND yNext >= 0 AND GVL.board[xNext,yNext].isEmpty) THEN
		selectedPiece.validMoveArr[xNext,yNext] := TRUE;
		temp := findPieceAtGivenLocation(x+1,y-1);
		jumpedPieceIndex := temp[1];
		IF(push(0, jumpedPieceIndex, xNext, yNext)) THEN
			//selectedPiece := checkForJumpBlack2(selectedPiece, selectedPieceIndex, xNext, yNext);
			selectedPiece := pop(selectedPiece, 1);
		END_IF
	END_IF
END_IF

// checks down and left
IF(x-1 >= 0 AND y-1 >= 0 AND NOT GVL.board[x-1,y-1].isEmpty AND GVL.board[x-1,y-1].isRed) THEN
	xNext := x - 2; // location of the space you could possibly jump to
	yNext := y - 2; // location of the space you could possibly jump to
	IF(xNext >= 0 AND yNext >= 0 AND GVL.board[xNext,yNext].isEmpty) THEN
		selectedPiece.validMoveArr[xNext,yNext] := TRUE;
		temp := findPieceAtGivenLocation(x-1,y-1);
		jumpedPieceIndex := temp[1];
		IF(push(0, jumpedPieceIndex, xNext, yNext)) THEN
			//selectedPiece := checkForJumpBlack2(selectedPiece, selectedPieceIndex, xNext, yNext);
			selectedPiece := pop(selectedPiece, 1);
		END_IF
	END_IF
END_IF

// checks up and left (FOR KINGS ONLY)
IF(x-1 < 8 AND y+1 >= 0 AND NOT GVL.board[x-1,y+1].isEmpty AND GVL.board[x-1,y+1].isRed AND selectedPiece.isKing) THEN
	xNext := x - 2; // location of the space you could possibly jump to
	yNext := y + 2; // location of the space you could possibly jump to		
	IF(xNext < 8 AND yNext >= 0 AND GVL.board[xNext,yNext].isEmpty) THEN
		selectedPiece.validMoveArr[xNext,yNext] := TRUE;
		temp := findPieceAtGivenLocation(x-1,y+1);
		jumpedPieceIndex := temp[1];
		IF(push(0, jumpedPieceIndex, xNext, yNext)) THEN
			//selectedPiece := checkForJumpBlack2(selectedPiece, selectedPieceIndex, xNext, yNext);
			selectedPiece := pop(selectedPiece, 1);
		END_IF
	END_IF
END_IF

// checks up and right (FOR KINGS ONLY)
IF(x+1 < 8 AND y+1 >= 0 AND NOT GVL.board[x+1,y+1].isEmpty AND GVL.board[x+1,y+1].isRed AND selectedPiece.isKing) THEN
	xNext := x + 2; // location of the space you could possibly jump to
	yNext := y + 2; // location of the space you could possibly jump to		
	IF(xNext < 8 AND yNext >= 0 AND GVL.board[xNext,yNext].isEmpty) THEN
		selectedPiece.validMoveArr[xNext,yNext] := TRUE;
		temp := findPieceAtGivenLocation(x+1,y+1);
		jumpedPieceIndex := temp[1];
		IF(push(0, jumpedPieceIndex, xNext, yNext)) THEN
			//selectedPiece := checkForJumpBlack2(selectedPiece, selectedPieceIndex, xNext, yNext);
			selectedPiece := pop(selectedPiece, 1);
		END_IF
	END_IF
END_IF

checkForJumpBlack4 := selectedPiece;


RETURN;

END_FUNCTION

// CODESYS_SoftMotion_Win_V3/Application/GameplayFunctions/ClearTakenPieces
PROGRAM ClearTakenPieces
VAR
	i : INT := 99;
	j : INT;
	k : INT;
	t : INT;
	currentRef : INT;
	found : BOOL;
END_VAR

IF(GVL.xMoveSpace <> -1 AND GVL.yMoveSpace <> -1) THEN
	i := 30;
	found := FALSE;
	WHILE(i >= 0 AND NOT found) DO
		
		
		// If the space identified in the jump move array and the space chosen match
		IF(GVL.jumpMoveArr[i].xMoveLocation = GVL.xMoveSpace AND GVL.jumpMoveArr[i].yMoveLocation = GVL.yMoveSpace) THEN
			found := TRUE;
			j := GVL.jumpMoveArr[i].jumpRef;
			k := i;
			WHILE(j >= 0 AND k >= 0) DO
				IF(GVL.jumpMoveArr[k].jumpRef = j) THEN					
					// Moves piece to its original location (off of the board)
					GVL.pieces[GVL.jumpMoveArr[k].jumpedPieceColor, GVL.jumpMoveArr[k].jumpedPieceIndex].translatedLocation[0] := 0;
					GVL.pieces[GVL.jumpMoveArr[k].jumpedPieceColor, GVL.jumpMoveArr[k].jumpedPieceIndex].translatedLocation[1] := 0;
						
					// Nulls out information for all taken pieces
					GVL.pieces[GVL.jumpMoveArr[k].jumpedPieceColor, GVL.jumpMoveArr[k].jumpedPieceIndex].isTaken := TRUE;	
					GVL.pieces[GVL.jumpMoveArr[k].jumpedPieceColor, GVL.jumpMoveArr[k].jumpedPieceIndex].isKing := FALSE;
					
					IF(GVL.board[GVL.jumpMoveArr[k].xJumpedLocation, GVL.jumpMoveArr[k].yJumpedLocation].isBlack) THEN
						GVL.blackPiecesTaken := GVL.blackPiecesTaken + 1;
					END_IF
					
					// Clears board space occupied by piece that was jumped
					GVL.board[GVL.jumpMoveArr[k].xJumpedLocation, GVL.jumpMoveArr[k].yJumpedLocation].isEmpty := TRUE;
					GVL.board[GVL.jumpMoveArr[k].xJumpedLocation, GVL.jumpMoveArr[k].yJumpedLocation].isRed := FALSE;
					GVL.board[GVL.jumpMoveArr[k].xJumpedLocation, GVL.jumpMoveArr[k].yJumpedLocation].isBlack := FALSE;
					
						
					// Sets pieces current location to invalid values
					GVL.pieces[GVL.jumpMoveArr[k].jumpedPieceColor, GVL.jumpMoveArr[k].jumpedPieceIndex].currentLocation[0] := -1;
					GVL.pieces[GVL.jumpMoveArr[k].jumpedPieceColor, GVL.jumpMoveArr[k].jumpedPieceIndex].currentLocation[1] := -1;
						
					// Nulls out pieces current valid move array
					GVL.pieces[GVL.jumpMoveArr[k].jumpedPieceColor, GVL.jumpMoveArr[k].jumpedPieceIndex].validMoveArr := GVL.noValidMoveArr;
					
					j := GVL.jumpMoveArr[k].lastJumpRef;
					
					WHILE(GVL.test) DO
								//
					END_WHILE
					
				END_IF
				k := k - 1;
			END_WHILE
		END_IF
		i := i - 1;
	END_WHILE
	(*FOR i := 0 TO 8 DO
		GVL.jumpMoveArr[i].numPiecesToJump := 0;
		GVL.jumpMoveArr[i].jumpedPieceColor := 0;
		GVL.jumpMoveArr[i].jumpedPieceIndex := 0;
		GVL.jumpMoveArr[i].xMoveLocation := 0;
		GVL.jumpMoveArr[i].yMoveLocation := 0;
	END_FOR*)
END_IF

END_PROGRAM

// CODESYS_SoftMotion_Win_V3/Application/GameplayFunctions/clearJumpArr
FUNCTION clearJumpArr : Bool
VAR_INPUT
END_VAR
VAR
	i : INT;
END_VAR

FOR i := 0 TO 99 DO
	GVL.jumpMoveArr[i].jumpedPieceColor := 0;
	GVL.jumpMoveArr[i].jumpedPieceIndex := 0;
	GVL.jumpMoveArr[i].jumpRef := 0;
	GVL.jumpMoveArr[i].lastJumpRef := -1;
	GVL.jumpMoveArr[i].numPiecesToJump := 0;
	GVL.jumpMoveArr[i].xJumpedLocation := 0;
	GVL.jumpMoveArr[i].xMoveLocation := 0;
	GVL.jumpMoveArr[i].yJumpedLocation := 0;
	GVL.jumpMoveArr[i].yMoveLocation := 0;
END_FOR

RETURN;

END_FUNCTION

// CODESYS_SoftMotion_Win_V3/Application/GameplayFunctions/MovePieceMotion
FUNCTION_BLOCK MovePieceMotion
VAR_INPUT
	xPos: LREAL;
	yPos: LREAL;
	zPos: LREAL;
	ExecuteMove: BOOL;
END_VAR
VAR_IN_OUT

END_VAR

VAR_OUTPUT
	
	MoveDone: BOOL;
END_VAR
VAR
	xMove : SM3_Basic.MC_MoveAbsolute;
	yMove : SM3_Basic.MC_MoveAbsolute;
	zMove : SM3_Basic.MC_MoveAbsolute;
	ExecuteInternal : BOOL;
END_VAR

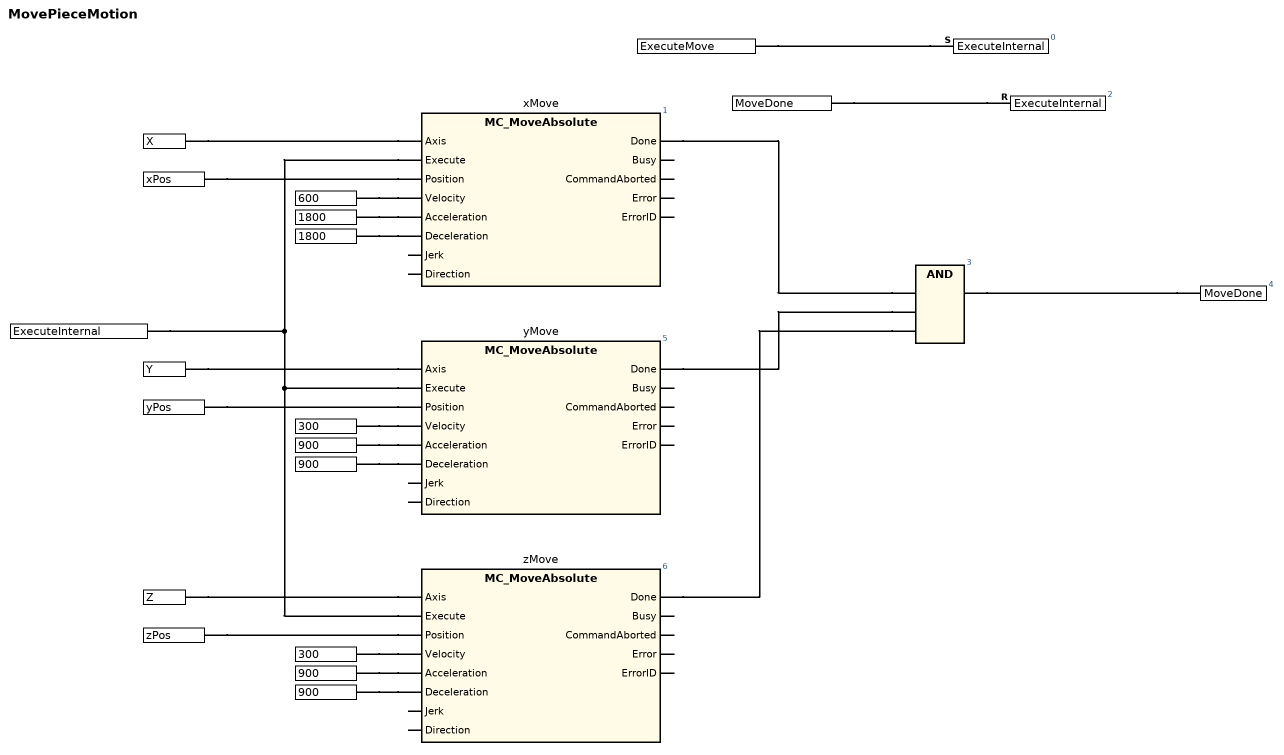
ExecuteInternal S= ExecuteMove;
xMove(
    Axis := X,
    Execute := ExecuteInternal,
    Position := xPos,
    Velocity := 600,
    Acceleration := 1800,
    Deceleration := 1800); // MC_MoveAbsolute
ExecuteInternal R= MoveDone;
MoveDone := xMove.Done AND yMove.Done AND zMove.Done;
yMove(
    Axis := Y,
    Execute := ExecuteInternal,
    Position := yPos,
    Velocity := 300,
    Acceleration := 900,
    Deceleration := 900); // MC_MoveAbsolute
zMove(
    Axis := Z,
    Execute := ExecuteInternal,
    Position := zPos,
    Velocity := 300,
    Acceleration := 900,
    Deceleration := 900); // MC_MoveAbsolute

END_FUNCTION_BLOCK

// CODESYS_SoftMotion_Win_V3/Application/GameplayFunctions/timeDelay
FUNCTION_BLOCK timeDelay
VAR_INPUT
	startTimer: BOOL;
END_VAR
VAR_OUTPUT
	done : BOOL;
END_VAR
VAR
	TON_0: TON;
END_VAR

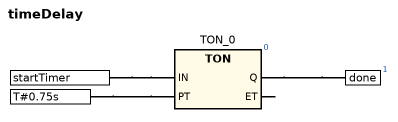
TON_0(IN := startTimer, PT := T#0.75s); // TON
done := TON_0.Q;

END_FUNCTION_BLOCK

// CODESYS_SoftMotion_Win_V3/Application/GameplayFunctions/AxisPositionFeedback
PROGRAM AxisPositionFeedback
VAR
	ReadPos: MC_GroupReadActualPosition;
	pos: SMC_POS_REF;
	enable: BOOL;
END_VAR

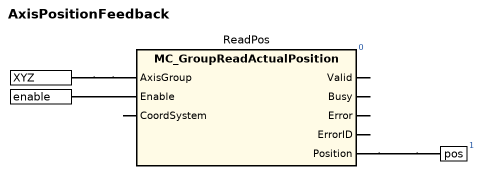
ReadPos(AxisGroup := XYZ, Enable := enable); // MC_GroupReadActualPosition
pos := ReadPos.Position;

END_PROGRAM

// CODESYS_SoftMotion_Win_V3/Application/JogFunctionality/JogLogic
PROGRAM JogLogic
VAR
	// Movement
	startup: BOOL := TRUE;
	
	xJogFwdPressed: BOOL;
	xJogRevPressed: BOOL;
	
	yJogFwdPressed: BOOL;
	yJogRevPressed: BOOL;
	
	zJogFwdPressed: BOOL;
	zJogRevPressed: BOOL;
END_VAR

// X_JogFwd := di_JogFwd AND NOT(di_JogBack); // From Will class

(* Startup *)
// System Reset Button
IF (TestPower.systemReset) THEN
	startup := TRUE;
	TestPower.systemReset := FALSE;
END_IF
// Startup Sequence
IF (startup) THEN
	GlobalVars.systemEnable := FALSE;
	xJogFwdPressed := FALSE;
	xJogRevPressed := FALSE;
	yJogFwdPressed := FALSE;
	yJogRevPressed := FALSE;
	zJogFwdPressed := FALSE;
	zJogRevPressed := FALSE;
	startup := FALSE;
	
	GlobalVars.p1Name := GlobalVars.p1DefaultName;
	GlobalVars.p2Name := GlobalVars.p2DefaultName;
	
	GlobalVars.xVel := 10;
	GlobalVars.xAcc := 100;
	GlobalVars.yVel := 10;
	GlobalVars.yAcc := 100;
	GlobalVars.zVel := 10;
	GlobalVars.zAcc := 100;
END_IF


(* System Disabled State Reset *)
IF (NOT GlobalVars.systemEnable) THEN
	GlobalVars.xJogFwd := FALSE;
	GlobalVars.xJogRev := FALSE;
	GlobalVars.yJogFwd := FALSE;
	GlobalVars.yJogRev := FALSE;
	GlobalVars.zJogFwd := FALSE;
	GlobalVars.zJogRev := FALSE;
	xJogFwdPressed := FALSE;
	xJogRevPressed := FALSE;
	yJogFwdPressed := FALSE;
	yJogRevPressed := FALSE;
	zJogFwdPressed := FALSE;
	zJogRevPressed := FALSE;
END_IF


(* Multitouch Precaution *)
IF (xJogFwdPressed AND xJogRevPressed) THEN
	xJogRevPressed := FALSE;
	xJogFwdPressed := FALSE;
END_IF
IF (yJogFwdPressed AND yJogRevPressed) THEN
	yJogRevPressed := FALSE;
	yJogFwdPressed := FALSE;
END_IF
IF (zJogFwdPressed AND zJogRevPressed) THEN
	zJogRevPressed := FALSE;
	zJogFwdPressed := FALSE;
END_IF


(* Jog Forward Button Pressed *)
// X Axis
IF (xJogFwdPressed) THEN
	IF (GlobalVars.systemEnable) THEN
		xJogRevPressed := FALSE;
		
		GlobalVars.xJogRev := FALSE;
		GlobalVars.xJogFwd := TRUE;		
	END_IF
END_IF
IF (NOT xJogFwdPressed) THEN
	GlobalVars.xJogFwd := FALSE;
END_IF
// Y Axis
IF (yJogFwdPressed) THEN
	IF (GlobalVars.systemEnable) THEN
		yJogRevPressed := FALSE;
		
		GlobalVars.yJogRev := FALSE;
		GlobalVars.yJogFwd := TRUE;		
	END_IF
END_IF
IF (NOT yJogFwdPressed) THEN
	GlobalVars.yJogFwd := FALSE;
END_IF
// Z Axis
IF (zJogFwdPressed) THEN
	IF (GlobalVars.systemEnable) THEN
		zJogRevPressed := FALSE;
		
		GlobalVars.zJogRev := FALSE;
		GlobalVars.zJogFwd := TRUE;		
	END_IF
END_IF
IF (NOT zJogFwdPressed) THEN
	GlobalVars.zJogFwd := FALSE;
END_IF


(* Jog Reverse Button Pressed *)
// X-Axis
IF (xJogRevPressed) THEN 
	IF (GlobalVars.systemEnable) THEN
		xJogFwdPressed := FALSE;
		GlobalVars.xJogFwd := FALSE;
		GlobalVars.xJogRev := TRUE;
	END_IF
END_IF
IF (NOT xJogRevPressed) THEN
	GlobalVars.xJogRev := FALSE;
END_IF
// Y Axis
IF (yJogRevPressed) THEN 
	IF (GlobalVars.systemEnable) THEN
		yJogFwdPressed := FALSE;
		GlobalVars.yJogFwd := FALSE;
		GlobalVars.yJogRev := TRUE;
	END_IF
END_IF
IF (NOT yJogRevPressed) THEN
	GlobalVars.yJogRev := FALSE;
END_IF
// Z Axis
IF (zJogRevPressed) THEN 
	IF (GlobalVars.systemEnable) THEN
		zJogFwdPressed := FALSE;
		GlobalVars.zJogFwd := FALSE;
		GlobalVars.zJogRev := TRUE;
	END_IF
END_IF
IF (NOT zJogRevPressed) THEN
	GlobalVars.zJogRev := FALSE;
END_IF

END_PROGRAM

// CODESYS_SoftMotion_Win_V3/Application/GameplayFunctions/SetupStart
PROGRAM SetupStart
VAR
	caseState: INT;
	SetupGo: BOOL;
	mover : MovePieceMotion;
	
	stop : BOOL;
	
	redStack0X : LREAL := 32.1;
	redStack0Y : LREAL := 159.8;
	
	blackStack0X : LREAL := 260.2;
	blackStack0Y : LREAL := 159.8;
	
	blackStackPos : INT := 3;
	blackStack : INT := 0;
	
	blackStackYDist : LREAL := -70;
	
	redStackPos : INT := 3;
	redStack : INT := 0;
	
	redStackYDist : LREAL := -70;
	
	pieceOffset : LREAL := 6.2;
	spaceOffset : LREAL := 20;
	
	pieceNumber : INT;
	colorNumber : INT;
	
	zUp : LREAL := 0;
	zDown : LREAL := 55;
	yOffset : LREAL := 18.3;
	xOffset : LREAL := 79.9;
	
	wait : timeDelay;
	
END_VAR

CASE caseState OF
	
000:
	IF(GVL.mechanicalSetup)THEN
		mover.zPos := zUp;
		caseState := 010;
	END_IF
	
010: 
	mover.ExecuteMove := TRUE;
	caseState := 011;

011: 
	IF(mover.MoveDone) THEN
		caseState := 012;
		mover.ExecuteMove := FALSE;
	END_IF
	
// Moves to the first position
012:
	mover.xPos := redStack0X;
	mover.yPos := redStack0Y + (redStack * redStackYDist);
	mover.zPos := zUp;
	caseState := 013;
	
013: 
	mover.ExecuteMove := TRUE;
	caseState := 014;

014: 
	IF(mover.MoveDone) THEN
		caseState := 015;
		mover.ExecuteMove := FALSE;
	END_IF
	
015:
	mover.zPos := zDown - ((4 - redStackPos) * pieceOffset);
	caseState := 016;

016: 
	mover.ExecuteMove := TRUE;
	caseState := 017;
	
017:
	IF(mover.MoveDone) THEN
		caseState := 018;
		mover.ExecuteMove := FALSE;
		GripperMove := TRUE;
		wait.startTimer := TRUE;
	END_IF
	
018:
	IF(wait.done)THEN
		wait.startTimer := FALSE;
		mover.zPos := zUp;
		caseState := 019;
	END_IF

019: 
	mover.ExecuteMove := TRUE;
	caseState := 020;
	
020:
	IF(mover.MoveDone)THEN
		caseState := 021;
		mover.ExecuteMove := FALSE;
	END_IF
	
021:
	mover.xPos := xOffset + (spaceOffset * GVL.pieces[colorNumber, pieceNumber].currentLocation[0]);
	mover.yPos :=  yOffset + (spaceOffset * GVL.pieces[colorNumber, pieceNumber].currentLocation[1]);
	mover.zPos := zUp;
	caseState := 022;
	
022:
	mover.ExecuteMove := TRUE;
	caseState := 023;
	
023:
	IF(mover.MoveDone)THEN
		caseState := 024;
		mover.ExecuteMove := FALSE;
	END_IF
		
024:
	mover.zPos := zDown;
	caseState := 025;

025: 
	mover.ExecuteMove := TRUE;
	caseState := 026;
	
026:
	IF(mover.MoveDone) THEN
		caseState := 027;
		mover.ExecuteMove := FALSE;
		GripperMove := FALSE;
		wait.startTimer := TRUE;
	END_IF
	
027:
	IF(wait.done)THEN
		wait.startTimer := FALSE;
		mover.zPos := zUp;
		caseState := 028;
	END_IF

028:
	mover.ExecuteMove := TRUE;
	caseState := 029;
	
029: 
	IF(mover.MoveDone)THEN
		caseState := 040;
		mover.ExecuteMove := FALSE;
	END_IF

040:
	redStackPos := redStackPos + 1;
	IF(redStackPos > 4)THEN
		redStack := redStack + 1;
		redStackPos := 0;
	END_IF
	IF(redStack > 3)THEN
		caseState := 049;
	ELSE
		pieceNumber := pieceNumber + 1;
		IF(pieceNumber > 11) THEN
			caseState := 049;
		ELSE
			caseState := 012;
		END_IF
		
	END_IF
	
049:
	colorNumber := 1;
	pieceNumber := 0;
	caseState := 050;
	
// Moves to the first position
050:
	mover.xPos := blackStack0X;
	mover.yPos := blackStack0Y + (blackStack * blackStackYDist);
	mover.zPos := zUp;
	caseState := 051;
	
051: 
	mover.ExecuteMove := TRUE;
	caseState := 052;

052: 
	IF(mover.MoveDone) THEN
		caseState := 053;
		mover.ExecuteMove := FALSE;
	END_IF
	
053:
	mover.zPos := zDown - ((4 - blackStackPos) * pieceOffset);
	caseState := 054;

054: 
	mover.ExecuteMove := TRUE;
	caseState := 055;
	
055:
	IF(mover.MoveDone) THEN
		caseState := 056;
		mover.ExecuteMove := FALSE;
		GripperMove := TRUE;
		wait.startTimer := TRUE;
	END_IF
	
056:
	IF(wait.done)THEN
		wait.startTimer := FALSE;
		mover.zPos := zUp;
		caseState := 057;
	END_IF

057: 
	mover.ExecuteMove := TRUE;
	caseState := 058;
	
058:
	IF(mover.MoveDone)THEN
		caseState := 059;
		mover.ExecuteMove := FALSE;
	END_IF
	
059:
	mover.xPos := xOffset + (spaceOffset * GVL.pieces[colorNumber, pieceNumber].currentLocation[0]);
	mover.yPos :=  yOffset + (spaceOffset * GVL.pieces[colorNumber, pieceNumber].currentLocation[1]);
	mover.zPos := zUp;
	caseState := 060;
	
060:
	mover.ExecuteMove := TRUE;
	caseState := 061;
	
061:
	IF(mover.MoveDone)THEN
		caseState := 062;
		mover.ExecuteMove := FALSE;
	END_IF
		
062:
	mover.zPos := zDown;
	caseState := 063;

063: 
	mover.ExecuteMove := TRUE;
	caseState := 064;
	
064:
	IF(mover.MoveDone) THEN
		caseState := 065;
		mover.ExecuteMove := FALSE;
		GripperMove := FALSE;
		wait.startTimer := TRUE;
	END_IF
	
065:
	IF(wait.done)THEN
		wait.startTimer := FALSE;
		mover.zPos := zUp;
		caseState := 066;
	END_IF

066:
	mover.ExecuteMove := TRUE;
	caseState := 067;
	
067: 
	IF(mover.MoveDone)THEN
		caseState := 070;
		mover.ExecuteMove := FALSE;
	END_IF

070:
	blackStackPos := blackStackPos + 1;
	IF(blackStackPos > 4)THEN
		blackStack := blackStack + 1;
		blackStackPos := 0;
	END_IF
	IF(blackStack > 3)THEN
		caseState := 100;
	ELSE
		pieceNumber := pieceNumber + 1;
		IF(pieceNumber > 11) THEN
			caseState := 100;
		ELSE
			caseState := 050;
		END_IF
		
	END_IF
	
	
	
100:
	GVL.mechanicalSetup := FALSE;
	IF(stop)THEN
		SetupGo := FALSE;
	END_IF
	
	
END_CASE

mover();
wait();

END_PROGRAM

// CODESYS_SoftMotion_Win_V3/Application/GameplayFunctions/CheckForWinner
PROGRAM CheckForWinner
VAR
	i : INT;
	redCounter : INT;
	blackCounter : INT;
END_VAR

redCounter := 0;
blackCounter := 0;

FOR i := 0 TO 11 DO 
	IF(GVL.pieces[0,i].isTaken)THEN
		redCounter := redCounter + 1;
	END_IF
END_FOR

FOR i := 0 TO 11 DO
	IF(GVL.pieces[1,i].isTaken)THEN
		blackCounter := blackCounter + 1;
	END_IF
END_FOR

// ALL THE BLACK PIECES ARE TAKEN, RED WINS
IF(blackCounter = 12) THEN
	GVL.redWins := TRUE;
END_IF

// ALL THE RED PIECES ARE TAKEN, BLACK WINS
IF(redCounter = 12) THEN
	GVL.blackWins := TRUE;
END_IF

END_PROGRAM

// CODESYS_SoftMotion_Win_V3/Application/GameplayFunctions/Teardown
PROGRAM Teardown
VAR
	currentPiece : INT;
	mover : MovePieceMotion;
	caseState: INT;
	
	
	redStack0X : LREAL := 32.1;
	redStack0Y : LREAL := 159.8;
	
	blackStack0X : LREAL := 260.2;
	blackStack0Y : LREAL := 159.8;
	
	blackStackYDist : LREAL := -70;
	
	redStackYDist : LREAL := -70;
	
	pieceOffset : LREAL := 6.2;
	spaceOffset : LREAL := 20;
	
	pieceNumber : INT;
	colorNumber : INT;
	
	zUp : LREAL := 0;
	zDown : LREAL := 55;
	yOffset : LREAL := 18.3;
	xOffset : LREAL := 79.9;
	
	wait : timeDelay;
	
	stop : BOOL;
	
END_VAR

CASE caseState OF
	
000: 
	IF(GVL.teardown) THEN
		caseState := 010;
	END_IF

// Move to up position
010:
	mover.zPos := zUp;
	caseState := 011;

011:
	mover.ExecuteMove := TRUE;
	caseState := 012;

012:
	IF(mover.MoveDone) THEN
		caseState := 013;
		mover.ExecuteMove := FALSE;
	END_IF
	
013:
	IF(GVL.pieces[0,currentPiece].currentLocation[0] = -1) THEN
		caseState := 013;
		currentPiece := currentPiece + 1;
		IF(currentPiece >= 12) THEN
			caseState := 050;
		END_IF
	ELSE
		mover.xPos := xOffset + (GVL.pieces[0,currentPiece].currentLocation[0] * spaceOffset);
		mover.yPos := yOffset + (GVL.pieces[0,currentPiece].currentLocation[1] * spaceOffset);
		mover.zPos := zUp;
		caseState := 014;		
	END_IF

014:
	mover.ExecuteMove := TRUE;
	caseState := 015;

015:
	IF(mover.MoveDone)THEN
		caseState := 016;
		mover.ExecuteMove := FALSE;
	END_IF

016:
	mover.zPos := zDown;
	caseState := 017;

017:
	mover.ExecuteMove := TRUE;
	caseState := 018;

018:
	IF(mover.MoveDone)THEN
		caseState := 019;
		mover.ExecuteMove := FALSE;
		GripperMove := TRUE;
		wait.startTimer := TRUE;
	END_IF
	
019:
	IF(wait.done)THEN
		caseState := 020;
		wait.startTimer := FALSE;
		mover.zPos := zUp;
	END_IF

020:
	mover.ExecuteMove := TRUE;
	caseState := 021;
	
021:
	IF(mover.MoveDone)THEN
		caseState := 022;
		mover.ExecuteMove := FALSE;
	END_IF

022:
	mover.xPos := redStack0X;
	mover.yPos := redStack0Y + (GVL.currentRedStack * redStackYDist);
	mover.zPos := zUp;
	caseState := 023;

023: 
	mover.ExecuteMove := TRUE;
	caseState := 024;
	
024:
	IF(mover.MoveDone)THEN
		caseState := 025;
		mover.ExecuteMove := FALSE;
	END_IF

025:
	mover.zPos := zDown - ((4 - GVL.currentRedStackPos) * pieceOffset);
	GVL.currentRedStackPos := GVL.currentRedStackPos - 1;
	IF(GVL.currentRedStackPos < 0) THEN
		GVL.currentRedStackPos := 4;
		GVL.currentRedStack := GVL.currentRedStack - 1;
	END_IF
	caseState := 026;

026:
	mover.ExecuteMove := TRUE;
	caseState := 027;
	
027:
	IF(mover.MoveDone) THEN
		mover.ExecuteMove := FALSE;
		caseState := 028;
		GripperMove := FALSE;
		wait.startTimer := TRUE;
	END_IF

028:
	IF(wait.done)THEN
		wait.startTimer := FALSE;
		mover.zPos := zUp;
		caseState := 029;
	END_IF

	
029:
	mover.ExecuteMove := TRUE;
	caseState := 030;

030:
	IF(mover.MoveDone) THEN
		mover.ExecuteMove := FALSE;
		currentPiece := currentPiece + 1;
		caseState := 013;
	END_IF
	
050:
	IF(stop)THEN
		caseState := 000;
	END_IF
	
END_CASE
mover();
wait();

END_PROGRAM

// CODESYS_SoftMotion_Win_V3/Application/Export/LogData
PROGRAM LogData
VAR
	filename: STRING := '/Windows/Logs/Log_HighCycleCount.csv';
	filehandle: SYSFILE.RTS_IEC_HANDLE;
	strMsg: STRING[255];
	FOResult: SYSFILE.RTS_IEC_RESULT;
	FWResult: SYSFILE.RTS_IEC_RESULT;
	FWStatus: POINTER TO RTS_IEC_RESULT;
	FCResult: SYSFILE.RTS_IEC_RESULT;
	bytesWritten: DWORD;
	bFileOpen: BOOL;
	iStatus : INT := 0;
	
	
	SafeToStop: BOOL;
	Result1: SYSFILE.RTS_IEC_RESULT;
	SizeFile: DWORD;
	ErrorID: INT;
	diActPosition: UDINT;
	
	LogIndex :DINT := 0;
	LogMsg : ARRAY [1..200] OF STRING[255];
	LogType : STRING;

	intIndex: DINT;
	
END_VAR

CASE iStatus OF
0: 
	IF(GVL.export)THEN
		iStatus := 1;
	END_IF
			

1: //Open File
	
	filehandle := SysFileOpen(szFile := filename, am := sysfile.AM_WRITE, pResult:= ADR(FOResult));
	IF (filehandle <> 16#00000000 AND filehandle <> 16#FFFFFFFF AND FOResult = cmperrors.Errors.ERR_OK) THEN 
		bFileOpen := TRUE;
		iStatus := iStatus + 1;
	ELSE
		ErrorID := -1 * iStatus;  //Open Memory Copy Failed
		iStatus := 99;
	END_IF//Open File

2:	//Log Data
	FOR intIndex := 1 TO LogIndex DO
		strMsg := LogMsg[intIndex];
		bytesWritten:= SysFileWrite(filehandle, ADR(strMsg), DINT_TO_DWORD(LEN(strMsg)), ADR(FWResult));
		IF FWResult <> CmpErrors.Errors.ERR_OK THEN
			ErrorID := -1 * iStatus;  //Log Data Failed
			iStatus := 100;
		END_IF
	END_FOR

3:  //Close File
	FCResult := SysFileClose(filehandle);
	IF FCResult = CmpErrors.Errors.ERR_OK THEN
		SafeToStop:=TRUE;
		iStatus := 0;
		GVL.export := FALSE;
	ELSE
		ErrorID := -1 * iStatus;  //File Close Failed
		iStatus := 99;
	END_IF
END_CASE

END_PROGRAM

// CODESYS_SoftMotion_Win_V3/Application/GameplayFunctions/boardSetup
PROGRAM boardSetup
VAR
	caseState: INT := 0;			//The case that is being intialized
	movePiece: MovePieceMotion;		//Instance of the MovePieceMotion, to move checkers
	gameReset: BOOL;				//Reset game board
	currentChecker: INT;			//Current checker being moved
	currentStack: INT;				//Current Stack where checkers are being pulled from
	currentColor: INT;				//Current Color of checkers that is being moved 
	currentStackPosition: INT;		//Currnet position within the stack that the checker is being pulled, 0 on top 4 on the bottom
	zUp: INT := 0;					//Z-axis all the way up position
	zDown: INT := 15;				//Z-axis all the way down position
	xStackOffset: LREAL; 			//Fill-in, this is the offset to the first stack from home
	xStackDistance: LREAL; 			//The X-axis distance between each stack
	yStackOffset: LREAL;			//Fill-in, this is the offset to the first stack from home
	yStackDistance: LREAL;			//The Y-axis distance between each stack
	pieceOffset: LREAL := 6.36;		//Height of one checker
	xBoardOffset: LREAL;			//X offset from home to the first square of the checker board
	yboardOffset: LREAL;			//Y offset from home to the first square of the checker board
	spaceOffset: LREAL := 20;				//Offset between each space on the checker board
	wait : timeDelay;				//Dwell to make sure that the grippers grip the checker piece
END_VAR

